(* CODESYS project CoDeSyS_Library_ST_MO
   Author: Razumovskiy
   Company: MechaTronics
   Description: Standart library for main typical devices
   LanguageModelAttribute: qualified-access-only
   Title: mt
   Version: 0.1.0.0

Project tree, tasks and I/O mapping:
  libraries: Standard, * (System)
  Drivers/
    FB_drv/
      function block drv_AI [ST]
      function block drv_AO [ST]
      function block drv_DI [ST]
      function block drv_DO [ST]
      function block drv_DOA [ST]
      function block drv_Flow [ST]
      function block drv_M [ST]
      function block drv_MR [ST]
      function block drv_V [ST]
    FB_sub/
      function sub_Axis_SP [ST]
      function block sub_Calibration [ST]
      function block sub_Filter [ST]
      function block sub_Slow [ST]
    UDT/
      data type AI_cfg
      data type AI_state
      data type AO_cfg
      data type AO_state
      data type Axis_cfg
      data type Axis_state
      data type DI_cfg
      data type DO_cfg
      data type DO_cfg_ext
      data type FE_cfg
      data type FE_state
      data type M_cfg
      data type M_state
      data type sub_Slow_cfg
      data type V_cfg
      data type V_state
    Union/
      uni/
        data type uni_AI_alarm
        data type uni_AI_cfg
        data type uni_AO_cfg
        data type uni_Axis_cfg
        data type uni_Axis_operation
        data type uni_DI_cfg
        data type uni_DO_cfg
        data type uni_FE_cfg
        data type uni_M_alarm
        data type uni_M_cfg
        data type uni_sub_Slow
        data type uni_V_alarm
        data type uni_V_cfg
      uni_udt/
        data type udt_AI_alarm
        data type udt_AI_cfg
        data type udt_AO_cfg
        data type udt_Axis_cfg
        data type udt_Axis_ErrorID
        data type udt_Axis_operation
        data type udt_DI_cfg
        data type udt_DO_cfg
        data type udt_FE_cfg
        data type udt_M_alarm
        data type udt_M_cfg
        data type udt_sub_Slow
        data type udt_V_alarm
        data type udt_V_cfg
  global variables sys
  System/
    FC/
      function drv_Alarm [ST]
      function drv_CMD [ST]
      function drv_Converter [ST]
      function drv_Scale [ST]
      function drv_Time_01S [ST]
      function drv_Time_C [ST]
      function drv_Time_R [ST]
      function drv_Time_S [ST]
      function drv_Time_X [ST]
    List/
      data type list_AI_SP
      data type list_Axis_SP
      data type list_Range
    UDT/
      data type Time_C
      data type Time_R
      data type Time_S
      data type Time_X
      data type udt_CMD
      data type udt_dev_list
      data type udt_DTL
      data type udt_state
      data type udt_Timer
      data type uni_CMD
      data type uni_dev_list
      data type uni_state
      data type uni_Timer
    program x00_Start [ST]
    program x99_End [ST]
  Информация библиотеки/
    function GetLibVersion [ST]
    function GetLibVersionNumber [ST]
    function IsLibReleased [ST]
*)

// Drivers/UDT/AI_cfg
TYPE AI_cfg :
STRUCT
	//configuration struct for Analog Inputs
		cfg				:uni_AI_cfg;	// HMI 0:	configuration word
		Input_Type		:INT := 1;		// HMI 1:	Input type: 0 = 0..20, 1 = 4..20, 2 = 0..10, 3 = Pt100, 4 = Pt1000
		Value_Type		:INT := 0;		// HMI 2:	Value type: 0 = %, 1 = Hz, 2 = l/h, etc
		Filter_Type		:INT := 1;		// HMI 3:	Execution clock for filter: 0 = every cycle of PLC, 1 = 0.1s, 2 = 1s
		Filter_Lim		:INT := 100;	// HMI 4:	Value of records in filter buffer
		Range			:list_Range;	// HMI 5:	Singal scale range
		Calibration		:REAL;			// HMI 13:	Static correction
		Multiplier		:REAL := 1;		// HMI 15:	Multiple correction
		SP				:list_AI_SP;	// HMI 17:	SP for limits
		T_SP			:ARRAY [0..3] OF INT;// HMI 26:	SP timers for limits
		ID				:INT;			// HMI 30:	ID for SCADA
		Name			:ARRAY [0..9] OF BYTE; // HMI 31:	Name
		ADDR			:INT;			// PLC xx:	address of inputs
		// HMI x - x is word number in shift address by start address
END_STRUCT
END_TYPE

// Drivers/UDT/AI_state
TYPE AI_state :
STRUCT
	//condition for Analog Inputs
		state		:uni_state;			// PLC 0:	condition word
		alarm		:uni_AI_alarm;		// HMI 1:	alarm word
		Status		:INT;				// HMI 2:	Status code for HMI
		Result		:REAL;				// HMI 3:	Result of convertation
		Signal		:REAL;				// HMI 5:	Input signal
		(*
			0 - disable
			1 - Result > L and Result < H
			2 - Result < L and Result > LL
			3 - Result > H and Result < HH
			4 - alarm "ST"
			5 - alarm "NC"
			6 - alarm LL
			7 - alarm HH
			
			if any alarm, than HMI will send message
		*)
END_STRUCT
END_TYPE

// Drivers/UDT/AO_cfg
TYPE AO_cfg :
STRUCT
	//configuration struct for Analog Outputs
		cfg				:uni_AO_cfg;	// HMI 0:	configuration word
		Output_Type		:INT := 1;		// HMI 1:	Output type: 0 = 0..20, 1 = 4..20, 2 = 0..10, 3 = Pt100, 4 = Pt1000
		Value_Type		:INT := 0;		// HMI 2:	Value type: 0 = %, 1 = Hz, 2 = l/h, etc
		Range			:list_Range;	// HMI 3:	Singal scale range
		SP_M			:REAL;			// HMI 10:	SP in manual mode
		ID				:INT;			// HMI 11:	ID for SCADA
		Name			:ARRAY [0..9] OF BYTE; // HMI 12:	Name
		ADDR			:INT;			// PLC xx:	address of inputs
END_STRUCT
END_TYPE

// Drivers/UDT/AO_state
TYPE AO_state :
STRUCT
	//condition for Analog Inputs
		state		:uni_state;			// HMI 0:	condition word
		Status		:INT;				// HMI 1:	Status code for HMI
		Result		:REAL;				// HMI 2:	Result of convertation
		Signal		:REAL;				// HMI 4:	Input signal
		(*
			0 - disable
			1 - activate
			
			if any alarm, than HMI will send message
		*)
END_STRUCT
END_TYPE

// Drivers/UDT/Axis_cfg
TYPE Axis_cfg :
STRUCT
	//configuration struct for Analog Inputs
		cfg				:uni_Axis_cfg;	// HMI 0:	configuration word
		Mode			:INT;			//	режим работы
		listSP			:list_Axis_SP;	//  уставки перемещения
		Direction		:BYTE := 1;
		posHome			:LREAL := 0.0;	//	уставка положения при калибровке нулевой точки
		ID				:INT;			// HMI 28:	ID for SCADA
		Name			:ARRAY [0..9] OF BYTE; // HMI 29:	Name
END_STRUCT
END_TYPE

// Drivers/UDT/Axis_state
TYPE Axis_state :
STRUCT
	//condition for Analog Inputs
		state		:uni_state;		// PLC 0:	condition word
		error		:uni_Axis_operation;// HMI 1:	alarm word
		busy		:uni_Axis_operation;
		done		:uni_Axis_operation;
		valid		:uni_Axis_operation;
		abort		:uni_Axis_operation;
		errorID		:udt_Axis_ErrorID;
		Status		:INT;				// HMI 2:	Status code for HMI
		Error_ID	:DWORD;				// HMI 3:	ErrorID
		Position	:LREAL;				// HMI 5:	Actual position
END_STRUCT
END_TYPE

// Drivers/UDT/DI_cfg
TYPE DI_cfg :
STRUCT
	cfg					:uni_DI_cfg;	// HMI 0:	configuration word
	//SP and another settings for Discrete Inputs
		SP_T_ON			:INT;			// HMI 1:	SP Time chatter filter starting, seconds
		SP_T_OFF		:INT;			// HMI 2:	SP Time chatter filter before stoping, seconds
END_STRUCT
END_TYPE

//History log:
//2023.01.10
//	1) data type 'bit' -> 'bool'
//	2) delete memory optimisation

// Drivers/UDT/DO_cfg
TYPE DO_cfg :
STRUCT
	cfg					:uni_DO_cfg;	// HMI 0:	configuration word
END_STRUCT
END_TYPE

// Drivers/UDT/DO_cfg_ext
TYPE DO_cfg_ext :
STRUCT
	cfg					:uni_DO_cfg;	// HMI 0:	configuration word
	//SP and another settings for Discrete Outputs
		SP_T			:REAL;			// HMI 1:	SP Time for impulse or PWM mode
		SP_A			:REAL;			// PLC 3:	SP % for PWM mode in auto mode
		SP_M			:REAL;			// PLC 5:	SP % for PWM mode in Manual mode
		SP_Min			:REAL := 10;	// PLC 7:	SP minimum value for switch on
		SP_Max			:REAL := 90;	// PLC 9:	SP value, while not switch off
END_STRUCT
END_TYPE

// Drivers/UDT/FE_cfg
TYPE FE_cfg :
STRUCT
	//configuration struct for FlowMeter
		cfg				:uni_FE_cfg;	// HMI 0:	configuration word
		Wieght			:REAL := 0.1;	// HMI 1:	Weight for 1 impulse
		Size_Wieght		:INT := 0;		// HMI 3:	Wieght of control unit - ml, l, m3
		Size_Time		:INT;			// HMI 5:	Speed of flow size: 0 - hour, 1 - minute, 2 - second
		Filter_Lim		:INT := 10;		// HMI 6:	Filter limit for summ values, max = 100
		Filter_Type		:INT;			// HMI 7:	Execution clock for filter: 0 = every cycle of PLC, 1 = 0.1s, 2 = 1s
		Clock			:INT := 1;		// HMI 8:	Cycle time for POU mode, ms
		Seans			:REAL;			// HMI 9:	Last seans data
		PreSP			:REAL;			// HMI 11:	PreSetpoint for one seans control
		SP				:REAL := 1;		// HMI 13:	Setpoint for one seans control
		DB				:REAL := 0.1;	// HMI 15:	Deadband for setpoint
		ID				:INT;			// HMI 17:	ID for SCADA
		Name			:ARRAY [0..9] OF BYTE; // HMI 18:	Name
		ADDR			:INT;			// PLC xx:	address of inputs
END_STRUCT
END_TYPE

// Drivers/UDT/FE_state
TYPE FE_state :
STRUCT
	//condition for Analog Inputs
		state		:uni_state;			// HMI 0:	condition word
		Status		:INT;				// HMI 1:	Status code for HMI
		Result		:REAL;				// HMI 2:	Actual flow speed
		AP			:REAL;				// HMI 4:	Actual flow value
		Last_AP		:REAL;				// HMI 6:	Last flow value
		(*
			0 - disable
			1 - Result > L and Result < H
			2 - Result < L and Result > LL
			3 - Result > H and Result < HH
			4 - alarm "ST"
			5 - alarm "NC"
			6 - alarm LL
			7 - alarm HH
			
			if any alarm, than HMI will send message
		*)
END_STRUCT
END_TYPE

// Drivers/UDT/M_cfg
TYPE M_cfg :
STRUCT
	cfg					:uni_M_cfg;		// HMI 0:	configuration word
	//SP and another settings for Motors
		SP_T_Delay_ON	:INT;			// HMI 1:	SP Time delay before starting, seconds
		SP_T_Delay_OFF	:INT;			// HMI 2:	SP Time delay before stoping, seconds
		SP_T_ON			:INT := 2;		// HMI 3:	SP Time feedback control during start, seconds
		SP_T_OFF		:INT := 2;		// HMI 4:	SP Time feedback control during stop, seconds
		ID				:INT;			// HMI 5:	ID for SCADA
		Name			:ARRAY [0..9] OF BYTE; // HMI 6:	Name
END_STRUCT
END_TYPE

//History log:
//2023.01.11
//	1) data type 'bit' -> 'bool'
//2023.01.18
//	1) delete service interval

// Drivers/UDT/M_state
TYPE M_state :
STRUCT
	state				:uni_state;			// HMI 0:	universal state word
	Alarm				:uni_M_alarm;		// HMI 1:	alarm word for Motors
	//specified condition for Motors	
		Status			:INT;				// HMI 2:	Status code for HMI
		(*
			0 - Successfully stopped
			1 - Successfully started
			2 - In the process of stopping
			3 - In the process of starting
			4 - Service maintance
			5 - alarm "No Ready"
			6 - alarm when stopping / now ON
			7 - alarm when starting / now OFF
			8 - alarm TS
			9 - alarm SF
			10 - alarm communication
			11 - External alarm
			99 - Emergency stop
			
			if any alarm, than device will try to stop
		*)
END_STRUCT
END_TYPE

//History log:
//2023.01.11
//	1) data type 'bit' -> 'bool'

// Drivers/UDT/sub_Slow_cfg
TYPE sub_Slow_cfg :
STRUCT
	cfg					:uni_sub_Slow;	// HMI 0:	configuration word
	//SP and another settings for sub driver Slow
		SP_Min			:REAL;
		SP_Max			:REAL;
		SP_Step_Up		:REAL;
		SP_Step_Down	:REAL;
		SP_T_Up			:REAL;
		SP_T_Down		:REAL;
END_STRUCT
END_TYPE

// Drivers/UDT/V_cfg
TYPE V_cfg :
STRUCT
	cfg					:uni_V_cfg;		// HMI 0:	configuration word
	//SP and another settings for Valves
		SP_T_Delay_ON	:INT;			// HMI 1:	SP Time delay before starting, seconds
		SP_T_Delay_OFF	:INT;			// HMI 2:	SP Time delay before stoping, seconds
		SP_T_ON			:INT := 10;		// HMI 3:	SP Time feedback control during start, seconds
		SP_T_OFF		:INT := 10;		// HMI 4:	SP Time feedback control during stop, seconds
		ID				:INT;			// HMI 5:	ID for SCADA
		Name			:ARRAY [0..9] OF BYTE; // HMI 6:	Name

END_STRUCT
END_TYPE

//History log:
//2023.01.13
//	1) data type 'bit' -> 'bool'
//	2) add TS, SF, SRV, Ext configurations
//	3) add SP_T_KM, fixed default SP time SP_T_ON/OFF '2 -> 10'

// Drivers/UDT/V_state
TYPE V_state :
STRUCT
	state				:uni_state;			// HMI 0:	universal state word
	Alarm				:uni_V_alarm;		// HMI 1:	alarm word for Valves
	//specified condition for Valves
		Status		:INT;					// HMI 2:	Status code for HMI
		(*
			0 - Successfully stopped
			1 - Successfully started
			2 - In the process of stopping
			3 - In the process of starting
			4 - Service maintance
			5 - alarm "No Ready"
			6 - alarm when opening / now ON
			7 - alarm when closing / now OFF
			8 - alarm TS
			9 - alarm SF
			10 - alarm communication
			11 - External alarm
			12 - alarm while opening / now close
			13 - alarm while opening / now no FB
			14 - alarm while closing / now open
			15 - alarm while closing / now no FB
			99 - Emergency stop
			
			if any alarm, than device will try to stop
		*)
END_STRUCT
END_TYPE

//History log:
//2023.01.11
//	1) data type 'bit' -> 'bool'

// System/List/list_AI_SP
TYPE list_AI_SP :
STRUCT
	HH			:REAL := 90;
	H			:REAL := 75;
	L			:REAL := 25;
	LL			:REAL := 10;
	SC			:REAL := 105;
	NC			:REAL := -5;
END_STRUCT
END_TYPE

// System/List/list_Axis_SP
TYPE list_Axis_SP :
STRUCT
	//configuration struct for axis movement
		Position				:LREAL := 0;	//Положение
		Velocity				:LREAL := 10;	//Скорость
		Acceleration			:LREAL := 10;	//Ускорение
		Deceleration			:LREAL := 10;	//Замедление
		C						:LREAL := 1;	//Коэффициент преобразования
END_STRUCT
END_TYPE

// System/List/list_Range
TYPE list_Range :
STRUCT
	Min_In		:REAL := 0;
	Max_In		:REAL := 100;
	Min_Out		:REAL := 0;
	Max_Out		:REAL := 100;
END_STRUCT
END_TYPE

// System/UDT/Time_C
TYPE Time_C :
STRUCT
	//control struct for a Timer Millisecond or counting
		CMD			:uni_Timer;		//command word
		SP			:REAL := 2.0;	//set point
		AP			:REAL;			//actual point
		One			:REAL := 0.1;	//impulse weight
		Percent		:REAL;			//progress 0..100%
		PT			:R_TRIG;		//control of a positive signal front
END_STRUCT
END_TYPE

// System/UDT/Time_R
TYPE Time_R :
STRUCT
	//control struct for a Timer High Accucary
		CMD			:uni_Timer;		//command word
		SP			:REAL := 2.000;	//set point as second
		AP			:REAL;			//actual point	
		RTC			:UDINT;			//real time stamp
		Delta		:UDINT;			//delta time control
		Percent		:REAL;			//progress 0..100%
END_STRUCT
END_TYPE

// System/UDT/Time_S
TYPE Time_S :
STRUCT
	//control struct for a Timer Second
		CMD			:uni_Timer;		//command word
		SP			:INT := 2;		//set point
		AP			:INT;			//actual point	
END_STRUCT
END_TYPE

// System/UDT/Time_X
TYPE Time_X :
STRUCT
	//control struct for a Timer High Accucary
		CMD			:uni_Timer;		//command word
		AP			:REAL;			//actual point	
		RTC			:UDINT;			//real time stamp
		Delta		:UDINT;			//delta time control
END_STRUCT
END_TYPE

// System/UDT/udt_CMD
TYPE udt_CMD :
STRUCT
	//standart control word
		Start_A 	:BIT;		// 0:	command for automatic control
		Start_M 	:BIT;		// 1:	command for manual control
		Manual		:BIT;		// 2:	mode of control (0 - automatic, 1 - manual (user or HMI))
		Lock		:BIT;		// 3:	technological lock
		Force		:BIT;		// 4:	forced control in manual mode
		Service		:BIT;		// 5:	activate service mode
		Local		:BIT;		// 6: 	activate local mode (0 - controlled by PLC, 1 - controlled by local keys)
		Reset		:BIT;		// 7:	resetting of device
		Alarm		:BIT;		// 8:	the device is in the alarm
		ResetOT		:BIT;		// 9:	reset opreational time
		Direction	:BIT;		// 10:	direction of moving
		LowSpeed	:BIT;		// 11:	low speed mode
		Test		:BIT;		// 12:	test run for once
		//you add more configuration bits for the project, if necessary, but not more than 15
END_STRUCT
END_TYPE

// System/UDT/udt_dev_list
TYPE udt_dev_list :
STRUCT
	//general types
		xDI		:BIT;		// 0:	any discrete input in *** mode or state
		xDO		:BIT;		// 1:	any discrete optput in *** mode or state
		xAI		:BIT;		// 2:	any analog input in *** mode or state
		xAO		:BIT;		// 3:	any analog ouput in *** mode or state
		xM		:BIT;		// 4:	any device type "M" in *** mode or state
		xV		:BIT;		// 5:	any device type "V" in *** mode or state
		xAxis	:BIT;		// 6:	any axis in *** mode or state
		Logick	:BIT;		// 7:	any logical block in *** mode or state
		xAny	:BIT;		// 8:	something input/output or device in *** mode or state
		xFE		:BIT;		// 9:	any flowmeter in *** mode or state
END_STRUCT
END_TYPE

// System/UDT/udt_DTL
TYPE udt_DTL :
STRUCT
	//Data Time List
		Year			:UINT;
		Month			:UINT;
		Day				:UINT;
		Hour			:UINT;
		Minute			:UINT;
		Second			:UINT;
		Millisecond		:UINT;
		WeekDay			:UINT;
		WeekYear		:UINT;
END_STRUCT
END_TYPE

// System/UDT/udt_state
TYPE udt_state :
STRUCT
	//unviversal condition word for any devices
		xON				:BIT;		// 0:	device succesfully started and working now
		xOFF			:BIT;		// 1:	device succesfulle stoped and stoping now
		Alarm			:BIT;		// 2:	device in something alarm
		Local			:BIT;		// 3:	device in local mode
		Service			:BIT;		// 4:	device in service mode
		warn_OT			:BIT;		// 5:	warning "Service maintenance is required, the interservice interval is exceeded"
		Pos_Ok			:BIT;		// 6:	position/speed reached or run now
		Ready			:BIT;		// 7:	device ready to start		
		Busy			:BIT;		// 8:	device busy and working now
		Done			:BIT;		// 9:	device finished task
		Enable			:BIT;		//10:	device enabled
		//you may add more configuration bits for the project, if necessary, but not more than 15
END_STRUCT
END_TYPE

// System/UDT/udt_Timer
TYPE udt_Timer :
STRUCT
	//configuration word for Timers
		Start		:BIT;			// 0:	Starting command
		Q			:BIT;			// 1:	Quit
		Pause		:BIT;			// 2:	Pause
		Reset		:BIT;			// 3:	Reset actual point to zero
		SFC			:BIT;			// 4:	Signal front control
		//you add more configuration bits for the project, if necessary, but not more than 16
END_STRUCT
END_TYPE

// System/UDT/uni_CMD
TYPE uni_CMD :
UNION
	//configuration word for Command Word
		hmi		:WORD;			//word for communication
		plc		:udt_CMD;	//tags for programming
END_UNION
END_TYPE

// System/UDT/uni_dev_list
TYPE uni_dev_list :
UNION
	//alarm word for device list
		hmi		:WORD;			//word for communication
		plc		:udt_dev_list;	//tags for programming
END_UNION
END_TYPE

// System/UDT/uni_state
TYPE uni_state :
UNION
	//universal state word
		hmi		:WORD;			//word for communication
		plc		:udt_state;		//tags for programming
END_UNION
END_TYPE

// System/UDT/uni_Timer
TYPE uni_Timer :
UNION
	//alarm word for Timers
		hmi		:WORD;			//word for communication
		plc		:udt_Timer;		//tags for programming
END_UNION
END_TYPE

// Drivers/Union/uni/uni_AI_alarm
TYPE uni_AI_alarm :
UNION
	//alarm word for Analog Inputs
		hmi		:WORD;			//word for communication
		plc		:udt_AI_alarm;	//tags for programming
END_UNION
END_TYPE

// Drivers/Union/uni/uni_AI_cfg
TYPE uni_AI_cfg :
UNION
	//configuration word for Analog Inputs
		hmi		:WORD;			//word for communication
		plc		:udt_AI_cfg;	//tags for programming
END_UNION
END_TYPE

// Drivers/Union/uni/uni_AO_cfg
TYPE uni_AO_cfg :
UNION
	//configuration word for Analog Inputs
		hmi		:WORD;			//word for communication
		plc		:udt_AO_cfg;	//tags for programming
END_UNION
END_TYPE

// Drivers/Union/uni/uni_Axis_cfg
TYPE uni_Axis_cfg :
UNION
	//configuration word forAxis
		hmi		:WORD;			//word for communication
		plc		:udt_Axis_cfg;	//tags for programming
END_UNION
END_TYPE

// Drivers/Union/uni/uni_Axis_operation
TYPE uni_Axis_operation :
UNION
	//modes word for Axis
		hmi		:WORD;			//word for communication
		plc		:udt_Axis_operation;	//tags for programming
END_UNION
END_TYPE

// Drivers/Union/uni/uni_DI_cfg
TYPE uni_DI_cfg :
UNION
	//configuration word for Discrete Inputs
		hmi		:WORD;			//word for communication
		plc		:udt_DI_cfg;	//tags for programming
END_UNION
END_TYPE

// Drivers/Union/uni/uni_DO_cfg
TYPE uni_DO_cfg :
UNION
	//configuration word for Discrete Outputs
		hmi		:WORD;			//word for communication
		plc		:udt_DO_cfg;	//tags for programming
END_UNION
END_TYPE

// Drivers/Union/uni/uni_FE_cfg
TYPE uni_FE_cfg :
UNION
	//configuration word for Analog Inputs
		hmi		:WORD;			//word for communication
		plc		:udt_FE_cfg;	//tags for programming
END_UNION
END_TYPE

// Drivers/Union/uni/uni_M_alarm
TYPE uni_M_alarm :
UNION
	//alarm word for Motors
		hmi		:WORD;			//word for communication
		plc		:udt_M_alarm;	//tags for programming
END_UNION
END_TYPE

// Drivers/Union/uni/uni_M_cfg
TYPE uni_M_cfg :
UNION
	//configuration word for Motors
		hmi		:WORD;			//word for communication
		plc		:udt_M_cfg;		//tags for programming
END_UNION
END_TYPE

// Drivers/Union/uni/uni_sub_Slow
TYPE uni_sub_Slow :
UNION
	//configuration word for sub driver Slow
		hmi		:WORD;			//word for communication
		plc		:udt_sub_Slow;	//tags for programming
END_UNION
END_TYPE

// Drivers/Union/uni/uni_V_alarm
TYPE uni_V_alarm :
UNION
	//alarm word for Valves
		hmi		:WORD;			//word for communication
		plc		:udt_V_alarm;	//tags for programming
END_UNION
END_TYPE

// Drivers/Union/uni/uni_V_cfg
TYPE uni_V_cfg :
UNION
	//configuration word for Valves
		hmi		:WORD;			//word for communication
		plc		:udt_V_cfg;		//tags for programming
END_UNION
END_TYPE

// Drivers/Union/uni_udt/udt_AI_alarm
TYPE udt_AI_alarm :
STRUCT
	//alarm word for Analog Inputs
		alm_ST		:BIT;		// 0:	alarm "No Ready" 
		alm_HH		:BIT;		// 1:	alarm "High alarm level"
		alm_H		:BIT;		// 2:	warning "High work level"
		alm_L		:BIT;		// 3:	warning "Low work level"
		alm_LL		:BIT;		// 4:	alarm "Low alarm level"
		alm_NC		:BIT;		// 5:	alarm "No connect"
		alm_SC		:BIT;		// 6:	alarm "Overload"
		//you add more configuration bits for the project, if necessary, but not more than 16
END_STRUCT
END_TYPE

// Drivers/Union/uni_udt/udt_AI_cfg
TYPE udt_AI_cfg :
STRUCT
	//configuration word for Analog Inputs
		use_Sim		:BIT;			// PLC 0:	0 - Normal mode of operation, 	1 - Simulation mode
		use_NoEmrg	:BIT;			// PLC 1:	0 - Use Emergency signal,		1 - Ignore Emergency signal
		use_RTD		:BIT := FALSE;	// HMI 2:	Use mode RTD/TC scaling
		use_Filter	:BIT := TRUE;	// HMI 3:	Use filter
		use_Light	:BIT;			// HMI 4:	Lighting status for screen indication
		use_Low		:BIT := TRUE;	// PLC 5:	Enable low level alarms
		use_High	:BIT := TRUE;	// PLC 6:	Enable high level alarms
		use_SC		:BIT;			// HMI 7:	use control wire break
		//you add more configuration bits for the project, if necessary, but not more than 16
END_STRUCT
END_TYPE

// Drivers/Union/uni_udt/udt_AO_cfg
TYPE udt_AO_cfg :
STRUCT
	//configuration word for Analog Outputs
		use_Sim		:BIT;			// PLC 0:	0 - Normal mode of operation, 	1 - Simulation mode
		use_NoEmrg	:BIT;			// HMI 1:	0 - Use Emergency signal,		1 - Ignore Emergency signal
		use_Light	:BIT;			// HMI 3:	Lighting status for screen indication
		//you add more configuration bits for the project, if necessary, but not more than 16
END_STRUCT
END_TYPE

// Drivers/Union/uni_udt/udt_Axis_cfg
TYPE udt_Axis_cfg :
STRUCT
	//configuration word for Analog Inputs
		use_Sim		:BIT;			// PLC 0:	0 - Normal mode of operation, 	1 - Simulation mode
		use_NoEmrg	:BIT;			// PLC 1:	0 - Use Emergency signal,		1 - Ignore Emergency signal
		use_Axis	:BIT;			// PLC 2: 	0 - Disable axis,				1 - Enable axis
		set_zero	:BIT;			// PLC 3:	0 - no activities,				1 - Set actual position as ZERO
		//you add more configuration bits for the project, if necessary, but not more than 16
END_STRUCT
END_TYPE

// Drivers/Union/uni_udt/udt_Axis_ErrorID
TYPE udt_Axis_ErrorID :
STRUCT
	//busy word for Axis
		read_position		:DWORD;		// 0:	MC_Position
		read_error			:DWORD;		// 1:	MC_ReadError
		reset_axis			:DWORD;		// 2:	MC_Reset
		power_on			:DWORD;		// 3:	MC_Power
		move_home			:DWORD;		// 4:	MC_Home
		move_jog			:DWORD;		// 5:	MC_Jog
		move_abs			:DWORD;		// 5:	MC_Abs
		move_vel			:DWORD;		// 7:	MC_Velocity
		set_pos				:DWORD;		// 8:	MC_SetPos
		tmp					:DWORD;		// 9:	temp value
		//you may add more configuration bits for the project, if necessary, but not more than 15
END_STRUCT
END_TYPE

// Drivers/Union/uni_udt/udt_Axis_operation
TYPE udt_Axis_operation :
STRUCT
	//busy word for Axis
		read_position		:BIT;		// 0:	MC_Position
		read_error			:BIT;		// 1:	MC_ReadError
		reset_axis			:BIT;		// 2:	MC_Reset
		power_on			:BIT;		// 3:	MC_Power
		move_home			:BIT;		// 4:	MC_Home
		move_jog			:BIT;		// 5:	MC_Jog
		move_abs			:BIT;		// 6:	MC_Abs
		move_vel			:BIT;		// 7:	MC_Velocity
		set_pos				:BIT;		// 8:	MC_SetPos
		ext					:BIT;		// 9:	external value
		tmp					:BIT;		//10:	temp value
		//you may add more configuration bits for the project, if necessary, but not more than 15
END_STRUCT
END_TYPE

// Drivers/Union/uni_udt/udt_DI_cfg
TYPE udt_DI_cfg :
STRUCT
	//configuration struct for Discrete Inputs
		use_Sim			:BIT;			// PLC 0:	0 - Normal mode of operation, 	1 - Simulation mode
		use_NoEmrg		:BIT;			// HMI 1:	0 - Use Emergency signal,		1 - Ignore Emergency signal
		use_NC			:BIT;			// HMI 2:	0 - Normal Open Signal, 		1 - Normal Close Signal
		use_Filter		:BIT;			// HMI 3:	0 - Not use filter,				1 - Use chatter filter
		//you may add more configuration bits for the project, if necessary, but not more than 15
END_STRUCT
END_TYPE

// Drivers/Union/uni_udt/udt_DO_cfg
TYPE udt_DO_cfg :
STRUCT
	//configuration struct for Discrete Outputs
		use_Sim			:BIT;			// PLC 0:	0 - Normal mode of operation, 	1 - Simulation mode
		use_NoEmrg		:BIT;			// HMI 1:	0 - Use Emergency signal,			1 - Ignore Emergency signal
		use_NC			:BIT;			// HMI 2:	0 - Normal Open Signal, 			1 - Normal Close Signal
		use_Impulse		:BIT;			// HMI 3:	0 - Permanent mode of operation, 	1 - Impulse mode of operation
		use_PWM			:BIT;			// HMI 4:	0 - Constant signal,				1 - PWM signal
		//you may add more configuration bits for the project, if necessary, but not more than 15
END_STRUCT
END_TYPE

// Drivers/Union/uni_udt/udt_FE_cfg
TYPE udt_FE_cfg :
STRUCT
	//configuration word for Analog Inputs
		use_Sim		:BIT;			// PLC 0:	0 - Normal mode of operation, 	1 - Simulation mode
		use_NoEmrg	:BIT;			// PLC 1:	0 - Use Emergency signal,		1 - Ignore Emergency signal
		use_POU		:BIT;			// HMI 2:	Call FE in special POU with fixed time
		use_Filter	:BIT := TRUE;	// HMI 3:	Use filter
		use_Light	:BIT;			// HMI 4:	Lighting status for screen indication
		use_DI		:BIT;			// HMI 5:	Use DI signal
		use_FM		:BIT;			// HMI 6:	Use weight control
		use_FM_Add	:BIT;			// HMI 7:	Use add weight control
		use_PreSP	:BIT := TRUE;	// HMI 8:	Use pre-SP  control
		use_SP		:BIT := TRUE;	// HMI 9:	Use SP control
		//you add more configuration bits for the project, if necessary, but not more than 16
END_STRUCT
END_TYPE

// Drivers/Union/uni_udt/udt_M_alarm
TYPE udt_M_alarm :
STRUCT
	//alarm word for Motors
		alm_QF			:BIT;		// 0:	alarm "No Ready" 
		alm_Start		:BIT;		// 1:	alarm "No In Work when starting"
		alm_Stop		:BIT;		// 2:	alarm "In Work when stopping"
		alm_TS			:BIT;		// 3:	alarm "No TS"
		alm_SF			:BIT;		// 4:	alarm "No Safety Signal"
		alm_Ext			:BIT;		// 5:	alarm "External alarm"
		alm_Link		:BIT;		// 6:	alarm communication
		alm_ES			:BIT;		// 7:	alarm "Emergency Stop"
		//you may add more configuration bits for the project, if necessary, but not more than 15
END_STRUCT
END_TYPE

// Drivers/Union/uni_udt/udt_M_cfg
TYPE udt_M_cfg :
STRUCT
	//configuration word for Motors
		use_Sim			:BIT;			// HMI 0:	0 - Normal mode of operation,	1 - Simulation mode
		use_NoEmrg		:BIT;			// HMI 1:	0 - Use Emergency signal,		1 - Ignore Emergency signal
		use_QF			:BIT := TRUE;	// HMI 2:	Feedback control "Ready"
		use_KM			:BIT := TRUE;	// HMI 3:	Feedback control "In work"
		use_Signal 		:BIT := TRUE;	// HMI 4:	Use external REQ
		//you may add more configuration bits for the project, if necessary, but not more than 15
END_STRUCT
END_TYPE

// Drivers/Union/uni_udt/udt_sub_Slow
TYPE udt_sub_Slow :
STRUCT
	//configuration struct for sub driver Slow
		//configuration word for Valves
		Enable			:BIT;			// HMI 0:	Enable algorythm
		use_Up			:BIT;			// HMI 1:	use slow mode for up value
		use_Down		:BIT;			// HMI 2:	use slow mode for down value
		use_Force_Up	:BIT;			// HMI 3:	use force mode for first up
		use_Force_Down	:BIT;			// HMI 4:	use force mode for last down
END_STRUCT
END_TYPE

// Drivers/Union/uni_udt/udt_V_alarm
TYPE udt_V_alarm :
STRUCT
	//alarm word for Valves
		alm_QF			:BIT;		// 0:	alarm "No Ready" 
		alm_Open		:BIT;		// 1:	alarm while opening
		alm_Close		:BIT;		// 2:	alarm while closing
		alm_Duo			:BIT;		// 3:	alarm duo signals FB_Open and FB_Close at once
		alm_TS			:BIT;		// 4:	alarm "No TS"
		alm_Ext			:BIT;		// 5:	alarm "External alarm"
		alm_Link		:BIT;		// 6:	alarm communication
		alm_ES			:BIT;		// 7:	alarm "Emergency Stop"
		//you may add more configuration bits for the project, if necessary, but not more than 15
END_STRUCT
END_TYPE

// Drivers/Union/uni_udt/udt_V_cfg
TYPE udt_V_cfg :
STRUCT
	//configuration struct for Valves
		//configuration word for Valves
		use_Sim			:BIT;			// HMI 0:	0 - Normal mode of operation,	1 - Simulation mode
		use_NoEmrg		:BIT;			// HMI 1:	0 - Use Emergency signal,		1 - Ignore Emergency signal
		use_QF			:BIT := TRUE;	// HMI 2:	Feedback control "Ready"
		use_FB_Open		:BIT := TRUE;	// HMI 3:	Feedback control "Valve Opened"
		use_FB_Close	:BIT := TRUE;	// HMI 4:	Feedback control "Valve Closed"
		use_CWF			:BIT := TRUE;	// HMI 5:	Close While Fault
		use_Air			:BIT;			// HMI 6:	Work mode for air valves
		use_Duo			:BIT;			// HMI 7:	Work mode for CW/CCW
		use_Once		:BIT;			// HMI 8:	Work mode without open/close feedback control after finishing movement
		use_Signal 		:BIT := TRUE;	// HMI 9:	Use external REQ
END_STRUCT
END_TYPE

// sys
{attribute 'qualified_only'}
VAR_GLOBAL
	//General management
		//Global controls
			All_Block		AT %MX0.0	:BOOL;				//Emergency stop
			All_Reset		AT %MX0.1	:BOOL;				//Reset all alarms
			All_Sim			AT %MX0.2	:BOOL;				//Switch simulation mode for all devices
			All_Auto		AT %MX0.3	:BOOL;				//Reset "CMD.plc.Manual" for all devices
			Silence			AT %MX0.4	:BOOL;				//Disable siren from HMI
			Save			AT %MX0.5	:BOOL;				//Save data to PVL
		//Service tags
			alm				AT %MW1		:uni_dev_list;		//Alarms flags for devices
			man				AT %MW2		:uni_dev_list;		//Manual flags for devices
			sim				AT %MW3		:uni_dev_list;		//Simulation flags for devices
			DTL				:udt_DTL;						//System time
			UpTime			:TIME;							//Work time after power on
			UpTime_ms		:UDINT;							//Work time after power on as millisecond
		//Global data
			LibVersion		AT %ML1		:VERSION;			//Version code
		
		//Additional tags and constans
			second			:REAL := (1.0/3600.0);	//wight of 1 second in hour format
			dev				:INT;					//device counter for FOR
			aws_ON			:BOOL := TRUE;			//always TRUE
			aws_OFF			:BOOL := FALSE;			//always FALSE
			StartUp_Load	:BOOL;		//First load configuration after power on
				
		//Impulse tags
			pulse_01s	:BOOL;					//global trigger 100 ms
			pulse_1s	:BOOL;					//global trigger 1 second
			
		//Clock tags
			clock_01s	:BOOL;					//global clock for 100 ms
			clock_05s	:BOOL;					//global clock for 500 ms
			clock_1s	:BOOL;					//global clock for 1 s
END_VAR

// System/x00_Start
PROGRAM x00_Start
VAR
	pulse_100ms			:UDINT;
	pulse_s				:UDINT;
	clock_100ms			:UDINT;
	clock_500ms			:UDINT;
	clock_s				:UDINT;
	support				:WORD;
	PT					:ARRAY [0..1] OF R_TRIG;
	NT					:ARRAY [0..1] OF F_TRIG;
END_VAR

//Read system time
	sys.UpTime := TIME();
	sys.UpTime_ms := TIME_TO_UDINT(sys.UpTime);
	
//Read library version
	sys.LibVersion := GetLibVersion();

//Pulse generation
	//pulse 100 ms
		IF (sys.UpTime_ms - pulse_100ms) >= 100 THEN
			sys.pulse_01s := TRUE;
			pulse_100ms := sys.UpTime_ms;
		else
			sys.pulse_01s := FALSE;
		END_IF;
	//pulse 1 s
		IF (sys.UpTime_ms - pulse_s) >= 1000 THEN
			sys.pulse_1s := TRUE;
			pulse_s := sys.UpTime_ms;
		else
			sys.pulse_1s := FALSE;
		END_IF;
		
//Clock generation
	//clock 100 ms
		IF (sys.UpTime_ms - clock_100ms) >= 100 THEN
			IF NOT sys.clock_01s THEN
				sys.clock_01s := TRUE;
			ELSE
				sys.clock_01s := FALSE;
			END_IF;
			clock_100ms := sys.UpTime_ms;
		END_IF;
		
	//clock 500 ms
		IF (sys.UpTime_ms - clock_500ms) >= 500 THEN
			IF NOT sys.clock_05s THEN
				sys.clock_05s := TRUE;
			ELSE
				sys.clock_05s := FALSE;
			END_IF;
			clock_500ms := sys.UpTime_ms;
		END_IF;
		
	//clock 1 s
		IF (sys.UpTime_ms - clock_s) >= 1000 THEN
			IF NOT sys.clock_1s THEN
				sys.clock_1s := TRUE;
			ELSE
				sys.clock_1s := FALSE;
			END_IF;
			clock_s := sys.UpTime_ms;
		END_IF;

END_PROGRAM

// Информация библиотеки/GetLibVersion
// This function has been automatically generated from the project information.
FUNCTION GetLibVersion : VERSION
VAR_INPUT
	
END_VAR

GetLibVersion.uiMajor := 0;
GetLibVersion.uiMinor := 1;
GetLibVersion.uiServicePack := 0;
GetLibVersion.uiPatch := 0;

END_FUNCTION

// System/x99_End
PROGRAM x99_End
VAR
END_VAR

//manual signal processing
	IF sys.man.plc.xAI OR sys.man.plc.xAO OR sys.man.plc.xDI OR sys.man.plc.xDO OR sys.man.plc.xM OR sys.man.plc.xV OR sys.man.plc.xAxis THEN
		sys.man.plc.xAny := TRUE;
	ELSE
		sys.man.plc.xAny := FALSE;
	END_IF;

//error signal processing
	IF sys.alm.plc.xAI OR sys.alm.plc.xM  OR sys.alm.plc.xV OR sys.alm.plc.xAxis OR sys.alm.plc.Logick THEN
		sys.alm.plc.xAny := TRUE;
	ELSE
		sys.alm.plc.xAny := FALSE;
	END_IF;
	
//simulation signal processing
	IF sys.sim.plc.xDO OR sys.sim.plc.xAO  OR sys.sim.plc.xM OR sys.sim.plc.xV OR sys.sim.plc.xAxis THEN
		sys.sim.plc.xAny := TRUE;
	ELSE
		sys.sim.plc.xAny := FALSE;
	END_IF;
	
//reset alarm processing
	IF sys.All_Reset THEN
		sys.alm.plc.xDO := FALSE;
		sys.alm.plc.xAO := FALSE;
		sys.alm.plc.xM := FALSE;
		sys.alm.plc.xV := FALSE;
		sys.alm.plc.xAxis := FALSE;
		sys.alm.plc.xAI := FALSE;
		sys.alm.plc.xM := FALSE;
		sys.alm.plc.xV := FALSE;
		sys.alm.plc.Logick := FALSE;
		sys.All_Reset := FALSE;
		sys.Silence := FALSE;
	END_IF;

//reset auto
	IF sys.All_Auto THEN
		sys.man.plc.xAI := FALSE;
		sys.man.plc.xDI := FALSE;
		sys.man.plc.xM := FALSE;
		sys.man.plc.xV := FALSE;
		sys.man.plc.xAO := FALSE;
		sys.man.plc.xDO := FALSE;
		sys.All_Auto := FALSE;
	END_IF
	
//Save data to PVL
	IF sys.Save THEN
		sys.Save := FALSE;
	END_IF

END_PROGRAM

// Информация библиотеки/GetLibVersionNumber
// This function has been automatically generated from the project information.
FUNCTION GetLibVersionNumber : DWORD
VAR_INPUT
	
END_VAR

GetLibVersionNumber := 65536;

END_FUNCTION

// Информация библиотеки/IsLibReleased
// This function has been automatically generated from the project information.
FUNCTION IsLibReleased : BOOL
VAR_INPUT
	
END_VAR

IsLibReleased := FALSE;

END_FUNCTION

// Drivers/FB_drv/drv_AI
FUNCTION_BLOCK drv_AI
VAR_INPUT
	Signal			:REAL;			//Analog input signal from PLC
END_VAR	
VAR_IN_OUT
	CMD				:uni_CMD;		//Non-retain structure with command word
	cfg				:AI_cfg;		//Retain structure with settings
	state			:AI_state;		//Non-retain structure with states information
END_VAR
VAR_OUTPUT
	Result			:REAL;			//Signal from sensor
END_VAR
VAR
	Value			:REAL;			//tmp value for calculating 
	support			:WORD;			//internal command buffer
	alm				:ARRAY [0..3] OF BOOL;			//support word for transfer alarms
	cnt				:INT;			//internal counter
	PT				:ARRAY [0..1] OF R_TRIG;
	NT				:ARRAY [0..1] OF F_TRIG;
	Clock			:ARRAY [0..3] OF Time_S;
	Filter			:sub_Filter;
END_VAR

//ANALOG INPUT
//control of typical analog sensors
// - pressure
// - level
// - flowmeter
// - etc

//global commands
	//auto mode
		IF sys.All_Auto THEN
			CMD.plc.Manual := FALSE;
		END_IF;
	//global reset
		IF sys.All_Reset THEN
			CMD.plc.Reset := TRUE;
		END_IF
		
//convert data
	//input scaling
	drv_Scale(
		Value := Signal,
		Input_Type := cfg.Input_Type,
		Range := cfg.Range,
		Result => state.Signal);
		
//NC control
	IF cfg.Input_Type = 1 AND state.Signal < 2.5 AND cfg.cfg.plc.use_SC AND CMD.plc.Start_A THEN
		state.alarm.plc.alm_NC := TRUE;
	END_IF
	
//SC control
IF cfg.cfg.plc.use_SC AND CMD.plc.Start_A  THEN
	CASE cfg.Input_Type OF 
		0: 	IF state.Signal > 21.0 AND cfg.cfg.plc.use_SC THEN			//0..20 mA
				state.alarm.plc.alm_SC := TRUE;
			END_IF
		1: 	IF state.Signal > 21.0 AND cfg.cfg.plc.use_SC THEN			//4..20 mA
				state.alarm.plc.alm_SC := TRUE;
			END_IF
		2: 	IF state.Signal > 10.5 AND cfg.cfg.plc.use_SC THEN			//0..10 V
				state.alarm.plc.alm_SC := TRUE;
			END_IF
		3: 	IF state.Signal > 155.0 AND cfg.cfg.plc.use_SC THEN			//-150..+150 C
				state.alarm.plc.alm_SC := TRUE;
			END_IF
		4: 	IF state.Signal > 255.0 AND cfg.cfg.plc.use_SC THEN			//-150..+250 C
				state.alarm.plc.alm_SC := TRUE;
			END_IF
	END_CASE
end_if
	
//device control
// 	drv_CMD(Emergency := support.0,
// 			CMD := CMD);
	//manual mode flag
		IF CMD.plc.Manual THEN sys.man.plc.xAI := TRUE; END_IF;
		
//data convert to phisycal value scale
	drv_Converter(
		Signal := Signal,
		Range := cfg.Range,
		Result => Value);
		
//signal's filter
	Filter(
		Start := CMD.plc.Start_A AND cfg.cfg.plc.use_Filter,
		Signal := Value,
		Filter_Type := cfg.Filter_Type,
		Filter_Lim := cfg.Filter_Lim,
		Result => Result);
		
//no filtering mode
	IF NOT cfg.cfg.plc.use_Filter THEN
		Result := Value;
	END_IF
	
//signal's correction
	IF NOT CMD.plc.Start_A THEN
		Result := 0;
	ELSE
		Result := Result * cfg.Multiplier + cfg.Calibration;
	END_IF
	
//state signal transfer
	state.Result := Result;

//alarms without time control
	//ST
		IF state.alarm.plc.alm_NC OR state.alarm.plc.alm_SC AND cfg.cfg.plc.use_SC AND CMD.plc.Start_A THEN
			state.alarm.plc.alm_ST := TRUE;
		END_IF
	
//alarms with time control
	//HH
		drv_Alarm(
			Signal := (Result > cfg.SP.HH AND cfg.cfg.plc.use_High),
			Reset := (CMD.plc.Reset OR NOT CMD.plc.Start_A),
			Clock := Clock[0].CMD,
			Alarm := alm[0]);
		state.alarm.plc.alm_HH := alm[0];
	//H
		drv_Alarm(
			Signal := (Result > cfg.SP.H),
			Reset := (CMD.plc.Reset OR NOT CMD.plc.Start_A OR (Result < cfg.SP.H)),
			Clock := Clock[1].CMD,
			Alarm := alm[1]);
		state.alarm.plc.alm_H := alm[1];
	//L
		drv_Alarm(
			Signal := (Result < cfg.SP.L),
			Reset := (CMD.plc.Reset OR NOT CMD.plc.Start_A OR (Result > cfg.SP.L)),
			Clock := Clock[2].CMD,
			Alarm := alm[2]);
		state.alarm.plc.alm_L := alm[2];
	//LL
		drv_Alarm(
			Signal := (Result < cfg.SP.LL AND cfg.cfg.plc.use_Low),
			Reset := (CMD.plc.Reset OR NOT CMD.plc.Start_A),
			Clock := Clock[3].CMD,
			Alarm := alm[3]);
		state.alarm.plc.alm_LL := alm[3];

//global alarm
	IF (state.alarm.plc.alm_ST OR state.alarm.plc.alm_HH OR state.alarm.plc.alm_LL) AND CMD.plc.Start_A THEN
		state.state.plc.Alarm := TRUE;
		sys.alm.plc.xAI := TRUE;
		CMD.plc.Alarm := TRUE;
	END_IF
	
//reset
	IF CMD.plc.Reset THEN
		state.alarm.hmi := 0;
		FOR cnt := 0 TO 3 DO
			Clock[cnt].CMD.plc.Reset := TRUE;
		END_FOR
		state.alarm.plc.alm_HH := FALSE;
		state.alarm.plc.alm_LL := FALSE;
		state.alarm.plc.alm_SC := FALSE;
		state.alarm.plc.alm_ST := FALSE;
		state.state.plc.Alarm := FALSE;
		CMD.plc.Alarm := FALSE;
		CMD.plc.Reset := FALSE;
	END_IF
	
//global state
	IF CMD.plc.Start_A THEN
		state.state.plc.xON := TRUE;
		state.state.plc.xOFF := FALSE;
	ELSE
		state.state.plc.xON := FALSE;
		state.state.plc.xOFF := TRUE;
	END_IF
	
//HMI light
	IF cfg.cfg.plc.use_Light THEN
		IF CMD.plc.Start_A THEN state.Status := 1; END_IF
		IF NOT state.alarm.plc.alm_L AND NOT state.alarm.plc.alm_H THEN state.Status := 1; END_IF
		IF state.alarm.plc.alm_L AND NOT state.alarm.plc.alm_LL THEN state.Status := 2; END_IF
		IF state.alarm.plc.alm_H AND NOT state.alarm.plc.alm_HH THEN state.Status := 3; END_IF
		IF state.alarm.plc.alm_LL THEN state.Status := 4; END_IF
		IF state.alarm.plc.alm_HH THEN state.Status := 5; END_IF
		IF state.alarm.plc.alm_ST THEN state.Status := 6; END_IF
		IF NOT CMD.plc.Start_A THEN state.Status := 0; END_IF
	ELSE
		state.Status := 0;
	END_IF
	
//call timers
	FOR cnt := 0 TO 3 DO
		Clock[0].SP := cfg.T_SP[cnt];
		drv_Time_S (Clock[cnt]);
	END_FOR

END_FUNCTION_BLOCK

// System/FC/drv_Scale
FUNCTION drv_Scale : bool
VAR_INPUT
	Value			:REAL;			//Analog input signal from PLC
	Input_Type		:INT;			//Input type: 0 = 0..20, 1 = 4..20, 2 = 0..10, 3 = Pt100, 4 = Pt1000
	Range			:list_Range;	//Signal scale range
END_VAR
VAR_OUTPUT
	Result 			:REAL;			//Analog input in phisical value
END_VAR
VAR
	Type_Min		:REAL;			//Minimum limit
	Type_Max		:REAL;			//Maximum limit
	Type_Limit		:int := 4;		//Update type in cyclic
END_VAR

//configuration transfering	
CASE Input_Type OF
	0: Type_Min := 0.0; Type_Max := 20.0;
	1: Type_Min := 4.0; Type_Max := 20.0;
	2: Type_Min := 0.0; Type_Max := 10.0;
	3: Result := Value;
	4: Result := Value;
END_CASE

//calculate real input value
IF Input_Type < 3 THEN
	Result := (Type_Max - Type_Min) / (Type_Limit - 0.0) * Value + Type_Min;
END_IF

//update type in cycle increment
IF Input_Type > Type_Limit THEN Input_Type := 0; END_IF

END_FUNCTION

// System/FC/drv_CMD
FUNCTION drv_CMD : bool
VAR_INPUT
	Emergency		:BOOL;		//signal of All_Block and Safety conditions
END_VAR
VAR_IN_OUT
	CMD				:uni_CMD;	//standart command word
END_VAR

// Device mode determination
	IF NOT Emergency THEN
		//Normal mode
		IF NOT CMD.plc.Force THEN
			//No technological lock
			IF NOT CMD.plc.Lock AND NOT CMD.plc.Alarm AND NOT CMD.plc.Service THEN
				//No manual mode
				IF NOT CMD.plc.Manual THEN
					CMD.plc.Start_M := CMD.plc.Start_A;
				END_IF;
			ELSE
				//Technological lock or device alarm
				CMD.plc.Start_M := FALSE;
			END_IF;
		END_IF;
	ELSE
		//Emergency stop
		CMD.plc.Start_M := FALSE;
	END_IF;

END_FUNCTION

// System/FC/drv_Converter
FUNCTION drv_Converter : bool
VAR_INPUT
	Signal			:REAL;			//Analog input signal from PLC
	Range			:list_Range;	//Signal scale range
END_VAR
VAR_OUTPUT
	Result			:REAL;			//Convertation result
END_VAR
VAR
	inv				:BOOL;			//inverse range
	Range_In		:REAL;			//full input range
	Range_Out		:REAL;			//full value range
	RR_Scale		:REAL;			//range in to range out scale
	Value_Min		:REAL;			//actual minimum output value
	Value_Max		:REAL;			//actual maximum output value
	Buffer			:REAL;			//tmp value for calculating
END_VAR

//Диапазон входного сигнала
IF Range.Min_In >= 0 THEN
    Range_In := Range.Max_In - Range.Min_In;
ELSE
    Range_In := Range.Max_In + ABS(Range.Min_In);
END_IF;

//Диапазон выходного сигнала
inv := FALSE;
IF Range.Min_Out >= 0 AND Range.Max_Out >= 0 THEN
    IF Range.Max_Out > Range.Min_Out THEN
        Range_Out := Range.Max_Out - Range.Min_Out;
        Value_Min := Range.Min_Out;
        Value_Max := Range.Max_Out;
    END_IF;
    IF Range.Max_Out < Range.Min_Out THEN
        Range_Out := Range.Min_Out - Range.Max_Out;
        Value_Min := Range.Max_Out;
        Value_Max := Range.Min_Out;
		inv := TRUE;
    END_IF;
END_IF;
IF Range.Min_Out <= 0 AND Range.Max_Out >= 0 THEN
    Range_Out := Range.Max_Out + ABS(Range.Min_Out);
	Value_Min := Range.Min_Out;
    Value_Max := Range.Max_Out;
END_IF;
IF Range.Min_Out <= 0 AND Range.Max_Out <= 0 THEN
    Range_Out := ABS(Range.Max_Out) + ABS(Range.Min_Out);
	Value_Min := Range.Min_Out;
    Value_Max := Range.Max_Out;
END_IF;
IF Range.Min_Out >= 0 AND Range.Max_Out <= 0 THEN
    Range_Out := ABS(Range.Max_Out) + ABS(Range.Min_Out);
	Value_Min := Range.Max_Out;
    Value_Max := Range.Min_Out;
END_IF;

//Соотношение диапазонов
IF Range_Out <> 0 THEN
	RR_Scale := Range_In / Range_Out;
END_IF

//Линеаризация
IF RR_Scale <> 0 THEN
	Buffer := Signal / RR_Scale;
END_IF

//Коррекция
Buffer := Buffer + Value_Min;

//Инверсия
IF inv THEN
    Buffer := Value_Max - Buffer;
END_IF;

//Ограничение снизу
IF Buffer < Value_Min THEN
    Buffer := Value_Min;
END_IF;

//Ограничение сверху
IF Buffer > Value_Max THEN
    Buffer := Value_Max;
END_IF;

//Вывод значения
Result := Buffer;

END_FUNCTION

// System/FC/drv_Alarm
FUNCTION drv_Alarm : bool
VAR_INPUT
	Signal			:BOOL;		//alarm condition
	Reset			:BOOL;		//local reset command
END_VAR
VAR_IN_OUT
	Clock			:uni_Timer;
	Alarm			:BOOL;		//alarm signal
END_VAR

//Standart alarm control function
	//Conditions compelete
		IF Signal THEN
			Clock.plc.Start := TRUE;
		ELSE
			Clock.plc.Start := FALSE;
		END_IF
	//Alarm control
		IF Clock.plc.Q THEN
			Alarm := TRUE;
		END_IF
	//Alarm reset
		IF sys.All_Reset OR Reset THEN
			Clock.plc.Start := FALSE;
			Alarm := FALSE;
		END_IF

END_FUNCTION

// System/FC/drv_Time_S
FUNCTION drv_Time_S : bool
VAR_IN_OUT
	T			:Time_S;		//configuration and command struct for timer of seconds
END_VAR

// Timer with a multiplicity of 1 second
	IF T.CMD.plc.Start AND NOT T.CMD.plc.Reset THEN
		// Turn on
		IF T.AP < T.SP THEN
			IF NOT T.CMD.plc.Pause AND sys.pulse_1s THEN
				T.AP := T.AP + 1;
			END_IF;
			T.CMD.plc.Q := FALSE;
		ELSE
			// SP is achieved
			T.CMD.plc.Q := TRUE;
		END_IF;
	ELSE
		// Turn off and reset
		T.AP := 0;
		T.CMD.plc.Q := FALSE;
		T.CMD.plc.Reset := FALSE;
	END_IF;

END_FUNCTION

// Drivers/FB_sub/sub_Filter
FUNCTION_BLOCK sub_Filter
VAR_INPUT
	Start			:BOOL;		//Enable filter
	Signal			:REAL;		//Input value
	Filter_Type		:INT;		//Execution clock for filter: 0 = every cycle of PLC, 1 = 0.1s, 2 = 1s
	Filter_Lim 		:INT;		//Value of records in filter buffer
END_VAR
VAR_OUTPUT
	Result			:REAL;		//Median value for all measurments
END_VAR
VAR
	cnt				:INT;		//calculate actual measurments
	x				:INT;		//internal counter for shifting array elements
	exe				:BOOL;		//command to execution filtering cycle
	Summ			:REAL;		//Summary value of all array's values
	DATA			:ARRAY [0..100] OF REAL;
END_VAR

//limit
	IF Filter_Lim > 100 THEN
		Filter_Lim := 100;
	END_IF

//adding new entyty
IF Start AND (Filter_Type = 0 OR (Filter_Type = 1 AND sys.pulse_01s) OR (Filter_Type = 2 AND sys.pulse_1s)) THEN
    IF cnt < Filter_Lim THEN
        cnt := cnt + 1;
    END_IF;
	exe := TRUE;
ELSIF NOT Start THEN
	cnt := 0;
	Result := Signal;
END_IF;

//start cycle
IF exe THEN
	//read new value
	DATA[0] := Signal;
	Summ := 0.0;
	
	//limit values
	IF cnt > Filter_Lim THEN
		cnt := Filter_Lim;
	END_IF;
	
	//shifting array
	FOR x := Filter_Lim TO 1 BY -1 DO
		DATA[x] := DATA[x - 1];
		IF x <= cnt AND Start THEN
			Summ := Summ + DATA[x];
		END_IF;
	END_FOR;
	
	//calculate median values
	IF cnt > 0 THEN
		Result := Summ / cnt;
	ELSE
		Result := 0.0;
	END_IF;
	
	//end cycle
	exe := FALSE;
END_IF;

END_FUNCTION_BLOCK

// Drivers/FB_drv/drv_AO
FUNCTION_BLOCK drv_AO
VAR_INPUT
	Signal			:REAL;			//Control signal from algorythm
END_VAR	
VAR_IN_OUT
	CMD				:uni_CMD;		//Non-retain structure with command word
	cfg				:AO_cfg;		//Retain structure with settings
	state			:AO_state;		//Non-retain structure with states information
END_VAR
VAR_OUTPUT
	Result_R		:REAL;			//Analog output signal to PLC in REAL
	Result_I		:INT;			//Analog output signal to PLC in INT
END_VAR
VAR
	Value			:REAL;			//tmp value for calculating 
	support			:WORD;			//internal command buffer
	cnt				:INT;			//internal counter
	PT				:ARRAY [0..1] OF R_TRIG;
	NT				:ARRAY [0..1] OF F_TRIG;
	Filter			:sub_Filter;
END_VAR

//ANALOG OUTPUT
//control of typical analog command
// - Hz setpoint for motors
// - % setpoint for valves

//global commands
	//auto mode
		IF sys.All_Auto THEN
			CMD.plc.Manual := FALSE;
		END_IF;
	//global reset
		IF sys.All_Reset THEN
			CMD.plc.Reset := TRUE;
		END_IF
		
//convert data
	IF cfg.cfg.plc.use_NoEmrg THEN
		support.0 := FALSE;
	ELSE
		support.0 := sys.All_Block;
	END_IF
	
//device control
	drv_CMD(Emergency := support.0,
			CMD := CMD);
	//manual mode flag
		IF CMD.plc.Manual THEN sys.man.plc.xAO := TRUE; END_IF;
		IF NOT CMD.plc.Manual THEN
			cfg.SP_M := Signal;
		END_IF
	//disable
		IF NOT CMD.plc.Start_M THEN
			cfg.SP_M := 0;
		END_IF

//data convert to phisycal value scale
	drv_Converter(
		Signal := cfg.SP_M,
		Range := cfg.Range,
		Result => Value);
	
//convert data
	drv_Scale(
		Value := Value,
		Input_Type := cfg.Output_Type,
		Range := cfg.Range,
		Result => state.Signal);

//state signal transfer
	state.Result := Value;
	
//result
IF NOT cfg.cfg.plc.use_Sim THEN
	Result_R := Value;
	Result_I := REAL_TO_INT(Value);
ELSE
	Result_R := 0.0;
	Result_I := 0;
END_IF
	
//global state
	IF CMD.plc.Start_A THEN
		state.state.plc.xON := TRUE;
		state.state.plc.xOFF := FALSE;
	ELSE
		state.state.plc.xON := FALSE;
		state.state.plc.xOFF := TRUE;
	END_IF
	
//HMI light
	IF cfg.cfg.plc.use_Light THEN
		IF CMD.plc.Start_A THEN state.Status := 1; END_IF
		IF NOT CMD.plc.Start_A THEN state.Status := 0; END_IF
	ELSE
		state.Status := 0;
	END_IF
	
//reset
	IF CMD.plc.Reset THEN
		state.state.plc.Alarm := FALSE;
		CMD.plc.Alarm := FALSE;
		CMD.plc.Reset := FALSE;
	END_IF

END_FUNCTION_BLOCK

// Drivers/FB_drv/drv_DI
FUNCTION_BLOCK drv_DI
VAR_INPUT
	Signal			:BOOL;		//Physical input value, i.e. %IX0.6
END_VAR
VAR_IN_OUT
	CMD				:uni_CMD;	//Non-retain structure with command word
	cfg				:DI_cfg;	//Retain structure with settings
END_VAR
VAR_OUTPUT
	Result			:BOOL;		//Logical output value, used in algorythms
END_VAR
VAR
	Value			:BOOL;		//internal signal
	Clock			:ARRAY [0..1] OF Time_R;
END_VAR

//DIGITAL INPUT
//Signals from sensors, for example:
//	- keys
//	- sensors
//	- etc

//global commands
	//auto mode
		IF sys.All_Auto THEN
			CMD.plc.Manual := FALSE;
		END_IF;

//normal close mode
	IF cfg.cfg.plc.use_NC THEN
		Value := NOT Signal;
	ELSE
		Value := Signal;
	END_IF;
	
// chatter filter
	IF cfg.cfg.plc.use_Filter THEN
	//turn on
		IF cfg.SP_T_ON > 0 AND Value THEN
			Clock[1].CMD.plc.Start := TRUE;
			Clock[0].CMD.plc.Start := FALSE;
			IF Clock[1].CMD.plc.Q THEN
				CMD.plc.Start_A := Value;
			END_IF;
		ELSIF Value THEN
			CMD.plc.Start_A := TRUE;
			Clock[1].CMD.plc.Start := FALSE;
			Clock[0].CMD.plc.Start := FALSE;
		END_IF;
			
	//turn off
		IF cfg.SP_T_OFF > 0 AND NOT Value THEN
			Clock[1].CMD.plc.Start := FALSE;
			Clock[0].CMD.plc.Start := TRUE;
			IF Clock[0].CMD.plc.Q THEN
				CMD.plc.Start_A := Signal;
			END_IF;
		ELSIF NOT Value THEN
			CMD.plc.Start_A := FALSE;
			Clock[1].CMD.plc.Start := FALSE;
			Clock[0].CMD.plc.Start := FALSE;
		END_IF;
	ELSE
		CMD.plc.Start_A := Value;
	END_IF;

//device control
	drv_CMD(Emergency := FALSE,
		CMD := CMD);
	//manual mode flag
		IF CMD.plc.Manual THEN sys.man.plc.xDI := TRUE; END_IF;

//result for main logic
	Result := CMD.plc.Start_M;

//call timers
	Clock[0].SP := INT_TO_REAL(cfg.SP_T_OFF);
	Clock[1].SP := INT_TO_REAL(cfg.SP_T_ON);
	drv_Time_R (Clock[0]);
	drv_Time_R (Clock[1]);

END_FUNCTION_BLOCK

// System/FC/drv_Time_R
FUNCTION drv_Time_R : bool
VAR_IN_OUT
	T			:Time_R;			//configuration and command struct for timer of milliseconds
END_VAR

// Timer with a multiplicity of 1 second
		
	//time counting
	IF T.CMD.plc.Start AND NOT T.CMD.plc.Reset THEN
		// Turn on
			IF T.RTC = 0 THEN
				T.RTC := sys.UpTime_ms;
			END_IF
		//delta calculate
			IF NOT T.CMD.plc.Q THEN
				T.Delta := sys.UpTime_ms - T.RTC;
			END_IF;
		//delta control
		IF T.AP < T.SP THEN
			T.CMD.plc.Q := FALSE;
		ELSE
			T.CMD.plc.Q := TRUE;
		END_IF;
	ELSE
		// Turn off and reset
		T.AP := 0;
		T.RTC := 0;
		T.Delta := 0;
		T.CMD.plc.Q := FALSE;
		T.CMD.plc.Reset := FALSE;
	END_IF;
	
	//convert data
		T.AP := UDINT_TO_REAL(T.Delta) / 1000;
	
	//calculate time
		IF T.SP > 0 AND T.CMD.plc.Start THEN
			T.Percent := (T.AP / T.SP) * 100.0;
		ELSE
			T.Percent := 0;
		END_IF;

END_FUNCTION

// Drivers/FB_drv/drv_DO
FUNCTION_BLOCK drv_DO
VAR_INPUT
	Signal			:BOOL;			//Command in automation mode from algorythms
END_VAR
VAR_IN_OUT
	CMD				:uni_CMD;		//Non-retain structure with command word
	cfg				:DO_cfg;		//Retain structure with settings
END_VAR
VAR_OUTPUT
	Result			:BOOL;			//Phisical output signal, i.e. %QX2.4
END_VAR
VAR
	support			:WORD;			//internal command buffer
	PT				:ARRAY [0..1] OF R_TRIG;
	NT				:ARRAY [0..1] OF F_TRIG;
END_VAR

//DIGITAL OUTPUT
//control of primitive devices, for example
// - solenoid valve
// - signal for data exchange with another device
// - etc

//global commands
	//auto mode
		IF sys.All_Auto THEN
			CMD.plc.Manual := FALSE;
		END_IF;
	//simulation mode
		PT[0](CLK := sys.All_Sim);
		NT[0](CLK := sys.All_Sim);
		IF PT[0].Q THEN cfg.cfg.plc.use_Sim := TRUE; END_IF;
		IF NT[0].Q THEN cfg.cfg.plc.use_Sim := FALSE; END_IF;
		if cfg.cfg.plc.use_Sim then sys.sim.plc.xDI := TRUE; end_if;

//convert data
	CMD.plc.Start_A := Signal;
	IF cfg.cfg.plc.use_NoEmrg THEN
		support.0 := FALSE;
	ELSE
		support.0 := sys.All_Block;
	END_IF
	
//device control
	drv_CMD(Emergency := support.0,
		CMD := CMD);
	//manual mode flag
		IF CMD.plc.Manual THEN sys.man.plc.xDO := TRUE; END_IF;
		
//command transfer
	support.15 := CMD.plc.Start_M;

//normal close mode
	IF cfg.cfg.plc.use_NC AND NOT cfg.cfg.plc.use_Sim THEN
		Result := NOT support.15;
	ELSE
		Result := support.15;
	END_IF;
	
//simulation mode
	IF cfg.cfg.plc.use_Sim THEN
		Result := FALSE;
	END_IF;

END_FUNCTION_BLOCK

// Drivers/FB_drv/drv_DOA
FUNCTION_BLOCK drv_DOA
VAR_INPUT
	Signal			:BOOL;			//Command in automation mode from algorythms
END_VAR
VAR_IN_OUT
	CMD				:uni_CMD;		//Non-retain structure with command word
	cfg				:DO_cfg_ext;	//Retain structure with settings
END_VAR
VAR_OUTPUT
	Result			:BOOL;			//Phisical output signal, i.e. %QX2.4
END_VAR
VAR
	support			:WORD;			//internal command buffer
	cnt				:INT;			//internal counter
	PT				:ARRAY [0..1] OF R_TRIG;
	NT				:ARRAY [0..1] OF F_TRIG;
	Clock			:ARRAY [0..1] OF Time_R;
END_VAR

//DIGITAL OUTPUT
//control of primitive devices, for example
// - solenoid valve
// - signal for data exchange with another device
// - etc

//global commands
	//auto mode
		IF sys.All_Auto THEN
			CMD.plc.Manual := FALSE;
		END_IF;
	//simulation mode
		PT[0](CLK := sys.All_Sim);
		NT[0](CLK := sys.All_Sim);
		IF PT[0].Q THEN cfg.cfg.plc.use_Sim := TRUE; END_IF;
		IF NT[0].Q THEN cfg.cfg.plc.use_Sim := FALSE; END_IF;
		IF cfg.cfg.plc.use_Sim THEN sys.sim.plc.xDO := TRUE; END_IF;

//convert data
	CMD.plc.Start_A := Signal;
	IF cfg.cfg.plc.use_NoEmrg THEN
		support.0 := FALSE;
	ELSE
		support.0 := sys.All_Block;
	END_IF
	
//device control
	drv_CMD(Emergency := support.0,
		CMD := CMD);
	//manual mode flag
		IF CMD.plc.Manual THEN sys.man.plc.xDO := TRUE; END_IF;
		
//command transfer
	support.15 := CMD.plc.Start_M;
	IF NOT CMD.plc.Manual THEN
		cfg.SP_M := cfg.SP_A;
	END_IF
	
//timer control
	Clock[0].CMD.plc.Start := support.15;
	IF Clock[0].CMD.plc.Q THEN
		Clock[0].CMD.plc.Reset := TRUE;
	END_IF
	
//output control
	IF cfg.cfg.plc.use_PWM THEN
		IF support.15 THEN
			IF Clock[0].Percent < cfg.SP_M THEN
				support.14 := TRUE;
			ELSE
				support.14 := FALSE;
			END_IF
			IF Clock[0].Percent > cfg.SP_Max THEN
				support.14 := TRUE;
			END_IF
			IF Clock[0].Percent < cfg.SP_Min THEN
				support.14 := FALSE;
			END_IF
		ELSE
			support.14 := FALSE;
		END_IF
	ELSE
		support.14 := support.15;
	END_IF

//normal close mode
	IF cfg.cfg.plc.use_NC AND NOT cfg.cfg.plc.use_Sim THEN
		Result := NOT support.14;
	ELSE
		Result := support.14;
	END_IF;
	
//simulation mode
	IF cfg.cfg.plc.use_Sim THEN
		Result := FALSE;
	END_IF;
	
//call timers
	Clock[0].SP := cfg.SP_T;
	FOR cnt := 0 TO 1 DO
		drv_Time_R (Clock[cnt]);
	END_FOR

END_FUNCTION_BLOCK

// Drivers/FB_drv/drv_Flow
FUNCTION_BLOCK drv_Flow
VAR_INPUT
	Start			:BOOL;			//Start flow control
	Signal_DI		:BOOL;			//Discrete impulse from flowmeter
	Signal_AI		:REAL;			//Analog data from flowmeter
END_VAR	
VAR_IN_OUT
	CMD				:uni_CMD;		//Non-retain structure with command word
	cfg				:FE_cfg;		//Retain structure with settings
	state			:FE_state;		//Non-retain structure with states information
END_VAR
VAR_OUTPUT
	PreDone			:BOOL;			//PreSP reached
	Done			:BOOL;			//SP reached
	Result			:REAL;			//Signal from flowmeter
END_VAR
VAR
	AP				:REAL;			//Actual time for countimng
	AP_POU			:REAL;			//Last actual value for counting
	SW				:REAL;			//Start weight for control 
	Value			:REAL;			//tmp value for calculating 
	support			:WORD;			//internal command buffer
	cnt				:INT;			//internal counter
	PT				:ARRAY [0..1] OF R_TRIG;
	NT				:ARRAY [0..1] OF F_TRIG;
	Clock			:ARRAY [0..1] OF Time_X;
	Filter			:sub_Filter;
END_VAR

//FLOWMETER
//control of typical flowmeter control
// - value of source product
// - flowspeed
// - statistics
// - etc

//global commands
	//auto mode
		IF sys.All_Auto THEN
			CMD.plc.Manual := FALSE;
		END_IF;
	//global reset
		IF sys.All_Reset THEN
			CMD.plc.Reset := TRUE;
		END_IF
		
//device control
	CMD.plc.Start_A := Start;
	drv_CMD(Emergency := support.0,
			CMD := CMD);
	//manual mode flag
		IF CMD.plc.Manual THEN sys.man.plc.xFE := TRUE; END_IF;
	//reset counter
		PT[1](CLK := CMD.plc.Start_M);
		IF PT[1].Q THEN
			state.Last_AP := state.AP;
			state.AP := 0.0;
		END_IF

//impulse mode
	PT[0](CLK := Signal_DI);
	IF cfg.cfg.plc.use_DI AND NOT cfg.cfg.plc.use_FM THEN
		IF NOT cfg.cfg.plc.use_POU THEN
			//time reset
			IF PT[0].Q THEN
				Clock[0].CMD.plc.Reset := TRUE;
				AP := Clock[0].AP;
			END_IF 
			//time control
			Clock[0].CMD.plc.Start := CMD.plc.Start_M;
		ELSE
			IF NOT PT[0].Q THEN
				AP_POU := AP_POU + cfg.Clock;
				AP := AP_POU;
			ELSE
				AP_POU := 0;
			END_IF
		END_IF
	ELSE
		Clock[0].CMD.plc.Start := FALSE;
	END_IF
	
//signal's filter
	IF cfg.cfg.plc.use_DI THEN
		//discrete input filtering
		IF PT[0].Q THEN
			Filter(
				Start := CMD.plc.Start_M,
				Signal := AP,
				Filter_Type := 0,
				Filter_Lim := cfg.Filter_Lim,
				Result => Result);
		END_IF
	ELSE
		//analog input filtering
		Filter(
			Start := CMD.plc.Start_M AND cfg.cfg.plc.use_Filter,
			Signal := Signal_AI,
			Filter_Type := cfg.Filter_Type,
			Filter_Lim := cfg.Filter_Lim,
			Result => Result);
		IF NOT cfg.cfg.plc.use_Filter THEN
			Result := Value;
		END_IF
	END_IF

//weight mode
	IF  cfg.cfg.plc.use_FM THEN
		IF NOT support.2 AND CMD.plc.Start_M THEN
			SW := Signal_AI;
			support.2 := TRUE;
		END_IF
		IF support.2 THEN
			IF NOT cfg.cfg.plc.use_FM_Add THEN
				AP := SW - Signal_AI;
			ELSE
				AP := Signal_AI - SW;
			END_IF
		END_IF
	END_IF
	
//state signal transfer
	state.Result := Result;
	
//summary flow control
	IF CMD.plc.Start_M THEN
		//flow actual calculating
		IF cfg.cfg.plc.use_DI THEN
			//for DI
			state.AP := state.AP + cfg.Wieght;
		ELSIF NOT cfg.cfg.plc.use_FM THEN
			//for AI
			IF sys.pulse_01s THEN
				CASE cfg.Size_Time OF
					0:	state.AP := state.AP + Result / 3600 / 10;
					1:	state.AP := state.AP + Result / 60 / 10;
					2:	state.AP := state.AP + Result / 10;
				END_CASE 
			END_IF 
		END_IF 
		//pre-setpoint control
		IF state.AP >= cfg.PreSP THEN
			state.state.plc.Pos_Ok := TRUE;
		END_IF
		//setpoint control
		IF (state.AP >= (cfg.SP - cfg.DB)) THEN
			state.state.plc.Done := TRUE;
		END_IF
	END_IF
	
//deactivate control
	NT[0](CLK := CMD.plc.Start_M);
	IF NT[0].Q THEN
		state.state.plc.Pos_Ok := FALSE;
		state.state.plc.Done := FALSE;
	END_IF
	
//global state
	IF CMD.plc.Start_M THEN
		state.state.plc.xON := TRUE;
		state.state.plc.xOFF := FALSE;
	ELSE
		state.state.plc.xON := FALSE;
		state.state.plc.xOFF := TRUE;
	END_IF
	
//HMI light
	IF cfg.cfg.plc.use_Light THEN
		IF CMD.plc.Start_M AND NOT state.state.plc.Pos_Ok THEN state.Status := 3; END_IF
		IF CMD.plc.Start_M AND state.state.plc.Pos_Ok AND NOT state.state.plc.Done THEN state.Status := 2; END_IF
		IF state.state.plc.Done THEN state.Status := 1; END_IF
		IF NOT CMD.plc.Start_M THEN state.Status := 0; END_IF
	ELSE
		state.Status := 0;
	END_IF
	
//data transfer
	PreDone := state.state.plc.Pos_Ok;
	Done := state.state.plc.Done;
	
//reset
	IF CMD.plc.Reset THEN
		state.state.plc.Alarm := FALSE;
		CMD.plc.Alarm := FALSE;
		CMD.plc.Reset := FALSE;
	END_IF
	
//call timers
	FOR cnt := 0 TO 1 DO
		drv_Time_X (Clock[cnt]);
	END_FOR

END_FUNCTION_BLOCK

// System/FC/drv_Time_X
FUNCTION drv_Time_X : bool
VAR_IN_OUT
	T			:Time_X;			//configuration and command struct for timer of milliseconds
END_VAR

// Timer with a multiplicity of 1 second
		
	//time counting
	IF T.CMD.plc.Start AND NOT T.CMD.plc.Reset THEN
		// Turn on
			IF T.RTC = 0 THEN
				T.RTC := sys.UpTime_ms;
				T.Delta := 0;
			END_IF
		//delta calculate
			IF NOT T.CMD.plc.Q THEN
				T.Delta := sys.UpTime_ms - T.RTC;
			END_IF;
	ELSE
		// Turn off and reset
		T.RTC := 0;
		T.CMD.plc.Q := FALSE;
		T.CMD.plc.Reset := FALSE;
	END_IF;
	
	//convert data
		T.AP := UDINT_TO_REAL(T.Delta) / 1000;

END_FUNCTION

// Drivers/FB_drv/drv_M
FUNCTION_BLOCK drv_M
VAR_INPUT
	Signal			:BOOL;			//Command in automation mode from algorythms
	FB_QF			:BOOL;			//Physical input value, control feedback signal 'Ready' or NOT 'Alarm'
	FB_KM			:BOOL;			//Physical input value, control feedback signal 'In Work' OR 'Run'
END_VAR
VAR_IN_OUT
	CMD				:uni_CMD;		//Non-retain structure with command word
	cfg				:M_cfg;			//Retain structure with settings
	state			:M_state;		//Non-retain structure with states information
END_VAR
VAR_OUTPUT
	CMD_FW			:BOOL;			//Phisical output signal for start device, i.e. %QX2.4
	CMD_Low			:BOOL;			//Phisical output signal for speed control, i.e. %QX2.7 - optional
	Done			:BOOL;			//Device in work
END_VAR
VAR
	support			:WORD;			//internal command buffer
	cnt				:INT;			//internal counter
	alm				:ARRAY [0..3] OF BOOL;			//support word for transfer alarms
	PT				:ARRAY [0..1] OF R_TRIG;
	NT				:ARRAY [0..1] OF F_TRIG;
	Clock			:ARRAY [0..3] OF Time_S;
END_VAR

//MOTORS
//control of typical motors
// - ventitalitons
// - pumps
// - conveyors
// - etc

//global commands
	//start device
		IF cfg.cfg.plc.use_Signal THEN
			CMD.plc.Start_A := Signal;
		END_IF
	//auto mode
		IF sys.All_Auto THEN
			CMD.plc.Manual := FALSE;
			CMD.plc.Force := FALSE;
		END_IF;
	//simulation mode
		PT[0](CLK := sys.All_Sim);
		NT[0](CLK := sys.All_Sim);
		IF PT[0].Q THEN cfg.cfg.plc.use_Sim := TRUE; END_IF;
		IF NT[0].Q THEN cfg.cfg.plc.use_Sim := FALSE; END_IF;
		if cfg.cfg.plc.use_Sim then sys.sim.plc.xM := TRUE; end_if;
	//global reset
		IF sys.All_Reset THEN
			CMD.plc.Reset := TRUE;
		END_IF

//convert data
	IF cfg.cfg.plc.use_NoEmrg THEN
		support.0 := FALSE;
	ELSE
		support.0 := sys.All_Block;
		IF support.0 THEN
			state.Alarm.plc.alm_ES := TRUE;
			state.Status := 99;
		END_IF
	END_IF

//alarms without time control
	//QF control
		IF cfg.cfg.plc.use_QF THEN
			IF NOT FB_QF THEN
				state.Alarm.plc.alm_QF := TRUE;
				state.Status := 5;
			END_IF
		END_IF
	
//device control
	drv_CMD(Emergency := support.0,
		CMD := CMD);
	//manual mode flag
		IF CMD.plc.Manual THEN sys.man.plc.xM := TRUE; END_IF;
		
//delay turn on
	IF cfg.SP_T_Delay_ON > 0 AND NOT CMD.plc.Manual THEN
		IF CMD.plc.Start_M THEN
			Clock[0].CMD.plc.Start := TRUE;
			Clock[1].CMD.plc.Start := FALSE;
			IF Clock[0].CMD.plc.Q THEN
				support.1 := TRUE;
			END_IF
		ELSE
			Clock[0].CMD.plc.Start := FALSE;
		END_IF
	ELSE
		support.1 := CMD.plc.Start_M;
	END_IF

//delay turn off
	IF cfg.SP_T_Delay_OFF > 0 AND NOT CMD.plc.Manual THEN
		IF NOT CMD.plc.Start_M THEN
			Clock[1].CMD.plc.Start := TRUE;
			Clock[0].CMD.plc.Start := FALSE;
			IF Clock[1].CMD.plc.Q THEN
				support.1 := FALSE;
			END_IF
		ELSE
			Clock[1].CMD.plc.Start := FALSE;
		END_IF
	ELSE
		support.1 := CMD.plc.Start_M;
	END_IF
	
//Starting
	IF support.1 AND state.Status < 4 AND NOT cfg.cfg.plc.use_Sim THEN
		support.2 := TRUE;
		support.3 := FALSE;
		IF cfg.cfg.plc.use_KM THEN
			//starting in progress
			IF NOT Clock[2].CMD.plc.Q AND NOT FB_KM THEN
				state.Status := 2;
			END_IF
			//starting in fault
			IF Clock[2].CMD.plc.Q AND NOT FB_KM THEN
				state.Status := 6;
			END_IF
			//starting complieted
			IF FB_KM AND state.Status < 4THEN
				state.Status := 1;
			END_IF
		ELSE
			//succesfuly started
			state.Status := 1;
		END_IF
	END_IF
	
//Stopping
	IF NOT support.1 AND NOT cfg.cfg.plc.use_Sim THEN
		support.2 := FALSE;
		support.3 := TRUE;
		IF cfg.cfg.plc.use_KM THEN
			//stoping in progress
			IF NOT Clock[3].CMD.plc.Q AND FB_KM THEN
				state.Status := 3;
			END_IF
			//stoping in fault
			IF Clock[3].CMD.plc.Q AND FB_KM THEN
				state.Status := 7;
			END_IF
			//stoping complieted
			IF NOT FB_KM AND state.Status < 4 THEN
				state.Status := 0;
			END_IF
		ELSE
			//succesfuly stopped
			state.Status := 0;
		END_IF
	END_IF
		
//alarms with time control
	//start alarm control
		drv_Alarm(
			Signal := (support.2 AND NOT FB_KM),
			Reset := (CMD.plc.Reset OR cfg.cfg.plc.use_Sim),
			Clock := Clock[2].CMD,
			Alarm := alm[0]);
		state.Alarm.plc.alm_Start := alm[0];
	//stop alarm control
		drv_Alarm(
			Signal := (support.3 AND FB_KM),
			Reset := (CMD.plc.Reset OR cfg.cfg.plc.use_Sim),
			Clock := Clock[3].CMD,
			Alarm := alm[1]);
		state.Alarm.plc.alm_Stop := alm[1];	

//global alarm
	IF (state.Status > 4 OR state.Alarm.hmi > 0) AND NOT cfg.cfg.plc.use_Sim THEN
		state.state.plc.Alarm := TRUE;
		sys.alm.plc.xM := TRUE;
		CMD.plc.Alarm := TRUE;
	END_IF
			
//reset
	IF CMD.plc.Reset THEN
		IF state.Status > 4 THEN
			state.Status := 0;
		END_IF
		FOR cnt := 0 TO 6 DO
			Clock[cnt].CMD.plc.Reset := TRUE;
		END_FOR
		state.state.plc.Alarm := FALSE;
		state.Alarm.hmi := 0;
		CMD.plc.Alarm := FALSE;
		CMD.plc.Reset := FALSE;
	END_IF
	
//Simulation
	IF cfg.cfg.plc.use_Sim THEN
		IF support.1 THEN
			state.Status := 1;
		ELSE
			state.Status := 0;
		END_IF
	END_IF

//ON & OFF
	IF (FB_KM OR (CMD.plc.Start_M AND (cfg.cfg.plc.use_Sim OR NOT cfg.cfg.plc.use_KM))) AND state.Status < 4 THEN
		state.state.plc.xON := TRUE;	
		state.state.plc.xOFF := FALSE;	
	ELSIF (NOT FB_KM OR (NOT CMD.plc.Start_M AND (cfg.cfg.plc.use_Sim OR NOT cfg.cfg.plc.use_KM)))AND state.Status < 4 THEN
		state.state.plc.xON := FALSE;	
		state.state.plc.xOFF := TRUE;
	ELSE
		state.state.plc.xON := FALSE;	
		state.state.plc.xOFF := FALSE;
	END_IF
	
//Done
	Done := state.state.plc.xON;

//commands
	//turn on
		IF support.2 AND NOT state.state.plc.Pos_Ok THEN
			CMD_FW := TRUE;
			IF CMD.plc.LowSpeed THEN
				CMD_Low := TRUE;
			ELSE
				CMD_Low := FALSE;
			END_IF
		END_IF
	//turn off
		IF support.3 AND NOT state.state.plc.Pos_Ok THEN
			CMD_FW := FALSE;
			CMD_Low := FALSE;
		END_IF
	//shutdown
		IF cfg.cfg.plc.use_Sim THEN
			CMD_FW := FALSE;
			CMD_Low := FALSE;
			CMD.plc.Reset := TRUE;
		END_IF
	
//call timers
	Clock[0].SP := cfg.SP_T_Delay_ON;
	Clock[1].SP := cfg.SP_T_Delay_OFF;
	Clock[2].SP := cfg.SP_T_ON;
	Clock[3].SP := cfg.SP_T_OFF;
	FOR cnt := 0 TO 3 DO
		drv_Time_S (Clock[cnt]);
	END_FOR

END_FUNCTION_BLOCK

// Drivers/FB_drv/drv_MR
FUNCTION_BLOCK drv_MR
VAR_INPUT
	Signal			:BOOL;			//Command in automation mode from algorythms
	FB_QF			:BOOL;			//Physical input value, control feedback signal 'Ready' or NOT 'Alarm'
	FB_KM			:BOOL;			//Physical input value, control feedback signal 'In Work' OR 'Run'
END_VAR
VAR_IN_OUT
	CMD				:uni_CMD;		//Non-retain structure with command word
	cfg				:M_cfg;		//Retain structure with settings
	state			:M_state;	//Non-retain structure with states information
END_VAR
VAR_OUTPUT
	CMD_FW			:BOOL;			//Phisical output signal for start device forward, i.e. %QX2.4
	CMD_RV			:BOOL;			//Phisical output signal for start device reverse, i.e. %QX2.4
	CMD_Low			:BOOL;			//Phisical output signal for speed control, i.e. %QX2.7 - optional
	Done			:BOOL;			//Device in work
END_VAR
VAR
	support			:WORD;			//internal command buffer
	cnt				:INT;			//internal counter
	alm				:ARRAY [0..3] OF BOOL;			//support word for transfer alarms
	PT				:ARRAY [0..1] OF R_TRIG;
	NT				:ARRAY [0..1] OF F_TRIG;
	Clock			:ARRAY [0..3] OF Time_S;
END_VAR

//MOTORS
//control of typical motors
// - ventitalitons
// - pumps
// - conveyors
// - etc

//global commands
	//start device
		IF cfg.cfg.plc.use_Signal THEN
			CMD.plc.Start_A := Signal;
		END_IF
	//auto mode
		IF sys.All_Auto THEN
			CMD.plc.Manual := FALSE;
		END_IF;
	//simulation mode
		PT[0](CLK := sys.All_Sim);
		NT[0](CLK := sys.All_Sim);
		IF PT[0].Q THEN cfg.cfg.plc.use_Sim := TRUE; END_IF;
		IF NT[0].Q THEN cfg.cfg.plc.use_Sim := FALSE; END_IF;
		IF cfg.cfg.plc.use_Sim THEN sys.sim.plc.xM := TRUE; END_IF;
	//global reset
		IF sys.All_Reset THEN
			CMD.plc.Reset := TRUE;
		END_IF

//convert data
	IF cfg.cfg.plc.use_NoEmrg THEN
		support.0 := FALSE;
	ELSE
		support.0 := sys.All_Block;
		IF support.0 THEN
			state.Alarm.plc.alm_ES := TRUE;
			state.Status := 99;
		END_IF
	END_IF

//alarms without time control
	//QF control
		IF cfg.cfg.plc.use_QF THEN
			IF NOT FB_QF THEN
				state.Alarm.plc.alm_QF := TRUE;
				state.Status := 5;
			END_IF
		END_IF
	
//device control
	drv_CMD(Emergency := support.0,
		CMD := CMD);
	//manual mode flag
		IF CMD.plc.Manual THEN sys.man.plc.xM := TRUE; END_IF;
		
//delay turn on
	IF cfg.SP_T_Delay_ON > 0 AND NOT CMD.plc.Manual THEN
		IF CMD.plc.Start_M THEN
			Clock[0].CMD.plc.Start := TRUE;
			Clock[1].CMD.plc.Start := FALSE;
			IF Clock[0].CMD.plc.Q THEN
				support.1 := TRUE;
			END_IF
		ELSE
			Clock[0].CMD.plc.Start := FALSE;
		END_IF
	ELSE
		support.1 := CMD.plc.Start_M;
	END_IF

//delay turn off
	IF cfg.SP_T_Delay_OFF > 0 AND NOT CMD.plc.Manual THEN
		IF NOT CMD.plc.Start_M THEN
			Clock[1].CMD.plc.Start := TRUE;
			Clock[0].CMD.plc.Start := FALSE;
			IF Clock[1].CMD.plc.Q THEN
				support.1 := FALSE;
			END_IF
		ELSE
			Clock[1].CMD.plc.Start := FALSE;
		END_IF
	ELSE
		support.1 := CMD.plc.Start_M;
	END_IF
	
//Starting
	IF support.1 AND state.Status < 4 AND NOT cfg.cfg.plc.use_Sim THEN
		support.2 := TRUE;
		support.3 := FALSE;
		IF cfg.cfg.plc.use_KM THEN
			//starting in progress
			IF NOT Clock[2].CMD.plc.Q AND NOT FB_KM THEN
				state.Status := 2;
			END_IF
			//starting in fault
			IF Clock[2].CMD.plc.Q AND NOT FB_KM THEN
				state.Status := 6;
			END_IF
			//starting complieted
			IF FB_KM AND state.Status < 4THEN
				state.Status := 1;
			END_IF
		ELSE
			//succesfuly started
			state.Status := 1;
		END_IF
	END_IF
	
//Stopping
	IF NOT support.1 AND NOT cfg.cfg.plc.use_Sim THEN
		support.2 := FALSE;
		support.3 := TRUE;
		IF cfg.cfg.plc.use_KM THEN
			//stoping in progress
			IF NOT Clock[3].CMD.plc.Q AND FB_KM THEN
				state.Status := 3;
			END_IF
			//stoping in fault
			IF Clock[3].CMD.plc.Q AND FB_KM THEN
				state.Status := 7;
			END_IF
			//stoping complieted
			IF NOT FB_KM AND state.Status < 4 THEN
				state.Status := 0;
			END_IF
		ELSE
			//succesfuly stopped
			state.Status := 0;
		END_IF
	END_IF

//alarms with time control
	//start alarm control
		drv_Alarm(
			Signal := (support.2 AND NOT FB_KM),
			Reset := (CMD.plc.Reset OR cfg.cfg.plc.use_Sim),
			Clock := Clock[2].CMD,
			Alarm := alm[0]);
		state.Alarm.plc.alm_Start := alm[0];
	//stop alarm control
		drv_Alarm(
			Signal := (support.3 AND FB_KM),
			Reset := (CMD.plc.Reset OR cfg.cfg.plc.use_Sim),
			Clock := Clock[3].CMD,
			Alarm := alm[1]);
		state.Alarm.plc.alm_Stop := alm[1];	
		
//global alarm
	IF (state.Status > 4 OR state.Alarm.hmi > 0) AND NOT cfg.cfg.plc.use_Sim THEN
		state.state.plc.Alarm := TRUE;
		sys.alm.plc.xM := TRUE;
		CMD.plc.Alarm := TRUE;
	END_IF
			
//reset
	IF CMD.plc.Reset THEN
		IF state.Status > 4 THEN
			state.Status := 0;
		END_IF
		FOR cnt := 0 TO 6 DO
			Clock[cnt].CMD.plc.Reset := TRUE;
		END_FOR
		state.state.plc.Alarm := FALSE;
		state.Alarm.hmi := 0;
		CMD.plc.Alarm := FALSE;
		CMD.plc.Reset := FALSE;
	END_IF
	
//Simulation
	IF cfg.cfg.plc.use_Sim THEN
		IF support.1 THEN
			state.Status := 1;
		ELSE
			state.Status := 0;
		END_IF
	END_IF

//ON & OFF
	IF (FB_KM OR (CMD.plc.Start_M AND (cfg.cfg.plc.use_Sim OR NOT cfg.cfg.plc.use_KM))) AND state.Status < 4 THEN
		state.state.plc.xON := TRUE;	
		state.state.plc.xOFF := FALSE;	
	ELSIF (NOT FB_KM OR (NOT CMD.plc.Start_M AND (cfg.cfg.plc.use_Sim OR NOT cfg.cfg.plc.use_KM)))AND state.Status < 4 THEN
		state.state.plc.xON := FALSE;	
		state.state.plc.xOFF := TRUE;
	ELSE
		state.state.plc.xON := FALSE;	
		state.state.plc.xOFF := FALSE;
	END_IF
	
//Done
	Done := state.state.plc.xON;

//commands
	//turn on
		IF support.2 AND NOT state.state.plc.Pos_Ok THEN
			IF NOT CMD.plc.Direction THEN
				CMD_FW := TRUE;
				CMD_RV := FALSE;
			ELSE
				CMD_FW := FALSE;
				CMD_RV := TRUE;
			END_IF
			IF CMD.plc.LowSpeed THEN
				CMD_Low := TRUE;
			ELSE
				CMD_Low := FALSE;
			END_IF
		END_IF
	//turn off
		IF support.3 AND NOT state.state.plc.Pos_Ok THEN
			CMD_FW := FALSE;
			CMD_RV := FALSE;
			CMD_Low := FALSE;
		END_IF
	//shutdown
		IF cfg.cfg.plc.use_Sim THEN
			CMD_FW := FALSE;
			CMD_RV := FALSE;
			CMD_Low := FALSE;
			CMD.plc.Reset := TRUE;
		END_IF
	
//call timers
	Clock[0].SP := cfg.SP_T_Delay_ON;
	Clock[1].SP := cfg.SP_T_Delay_OFF;
	Clock[2].SP := cfg.SP_T_ON;
	Clock[3].SP := cfg.SP_T_OFF;
	FOR cnt := 0 TO 3 DO
		drv_Time_S (Clock[cnt]);
	END_FOR

END_FUNCTION_BLOCK

// Drivers/FB_drv/drv_V
FUNCTION_BLOCK drv_V
VAR_INPUT
	Signal			:BOOL;			//Command in automation mode from algorythms
	FB_QF			:BOOL;			//Physical input value, control feedback signal 'Ready' or NOT 'Alarm'
	FB_Open			:BOOL;			//Physical input value, control feedback signal 'Open'
	FB_Close		:BOOL;			//Physical input value, control feedback signal 'Close'
END_VAR
VAR_IN_OUT
	CMD				:uni_CMD;		//Non-retain structure with command word
	cfg				:V_cfg;			//Retain structure with settings
	state			:V_state;		//Non-retain structure with states information
END_VAR
VAR_OUTPUT
	CMD_Open		:BOOL;			//Phisical output signal for opening, i.e. %QX2.4
	CMD_Close		:BOOL;			//Phisical output signal for closing, i.e. %QX2.5
	CMD_Low			:BOOL;			//Phisical output signal for speed control, i.e. %QX2.7 - optional
	Done			:BOOL;			//Device is open
END_VAR
VAR
	support			:WORD;
	cnt				:INT;			//internal counter
	alm				:ARRAY [0..3] OF BOOL;			//support word for transfer alarms
	PT				:ARRAY [0..3] OF R_TRIG;
	NT				:ARRAY [0..1] OF F_TRIG;
	Clock			:ARRAY [0..3] OF Time_S;
END_VAR

//VALVES
//control of typical air and electrical valves
// - doors
// - dampers
// - valves
// - etc

//global commands
	//start device
		IF cfg.cfg.plc.use_Signal THEN
			CMD.plc.Start_A := Signal;
		END_IF
	//auto mode
		IF sys.All_Auto THEN
			CMD.plc.Manual := FALSE;
			CMD.plc.Force := FALSE;
		END_IF;
	//simulation mode
		PT[0](CLK := sys.All_Sim);
		NT[0](CLK := sys.All_Sim);
		IF PT[0].Q THEN cfg.cfg.plc.use_Sim := TRUE; END_IF;
		IF NT[0].Q THEN cfg.cfg.plc.use_Sim := FALSE; END_IF;
		IF cfg.cfg.plc.use_Sim THEN sys.sim.plc.xV := TRUE; END_IF;
	//global reset
		IF sys.All_Reset THEN
			CMD.plc.Reset := TRUE;
		END_IF

//convert data
	IF cfg.cfg.plc.use_NoEmrg THEN
		support.0 := FALSE;
	ELSE
		support.0 := sys.All_Block;
		IF support.0 THEN
			state.Alarm.plc.alm_ES := TRUE;
			state.Status := 99;
		END_IF
	END_IF

//alarms without time control
	//QF control
		IF cfg.cfg.plc.use_QF THEN
			IF NOT FB_QF THEN
				state.Alarm.plc.alm_QF := TRUE;
				state.Status := 5;
			END_IF
		END_IF
	
//device control
	drv_CMD(Emergency := support.0,
		CMD := CMD);
	//manual mode flag
		IF CMD.plc.Manual THEN sys.man.plc.xV := TRUE; END_IF;
		
//delay turn on
	IF cfg.SP_T_Delay_ON > 0 AND NOT CMD.plc.Manual THEN
		IF CMD.plc.Start_M THEN
			Clock[0].CMD.plc.Start := TRUE;
			Clock[1].CMD.plc.Start := FALSE;
			IF Clock[0].CMD.plc.Q THEN
				support.1 := TRUE;
			END_IF
		ELSE
			Clock[0].CMD.plc.Start := FALSE;
		END_IF
	ELSE
		support.1 := CMD.plc.Start_M;
	END_IF

//delay turn off
	IF cfg.SP_T_Delay_OFF > 0 AND NOT CMD.plc.Manual THEN
		IF NOT CMD.plc.Start_M THEN
			Clock[1].CMD.plc.Start := TRUE;
			Clock[0].CMD.plc.Start := FALSE;
			IF Clock[1].CMD.plc.Q THEN
				support.1 := FALSE;
			END_IF
		ELSE
			Clock[1].CMD.plc.Start := FALSE;
		END_IF
	ELSE
		support.1 := CMD.plc.Start_M;
	END_IF
	
//Opening
	IF support.1 AND state.Status < 4 AND NOT cfg.cfg.plc.use_Sim THEN
		IF cfg.cfg.plc.use_Air THEN
			support.2 := TRUE;
		ELSIF NOT cfg.cfg.plc.use_Air AND (NOT FB_Open OR NOT cfg.cfg.plc.use_FB_Open) THEN
			support.2 := TRUE;
		ELSE
			support.2 := FALSE;
		END_IF
		support.3 := FALSE;
		Clock[2].CMD.plc.Start := TRUE;
		Clock[3].CMD.plc.Start := FALSE;
		IF cfg.cfg.plc.use_FB_Open THEN
			//opening in progress
			IF NOT Clock[2].CMD.plc.Q AND NOT FB_Open THEN
				state.Status := 2;
			END_IF
			//opening in fault
			IF Clock[2].CMD.plc.Q AND NOT FB_Open AND NOT state.state.plc.Pos_Ok THEN
				state.Status := 6;
			END_IF
			//opening complieted
			IF FB_Open THEN
				state.Status := 1;
			END_IF
		ELSE
			//succesfuly
			state.Status := 1;
		END_IF
	END_IF
	
//Closing
	IF NOT support.1 AND NOT cfg.cfg.plc.use_Sim THEN
		support.2 := FALSE;
		IF cfg.cfg.plc.use_Air THEN
			support.3 := TRUE;
		ELSIF NOT cfg.cfg.plc.use_Air AND (NOT FB_Close OR NOT cfg.cfg.plc.use_FB_Close) THEN
			support.3 := TRUE;
		ELSE
			support.3 := FALSE;
		END_IF
		Clock[2].CMD.plc.Start := FALSE;
		Clock[3].CMD.plc.Start := TRUE;
		IF cfg.cfg.plc.use_FB_Close THEN
			//opening in progress
			IF NOT Clock[3].CMD.plc.Q AND NOT FB_Close THEN
				state.Status := 3;
			END_IF
			//opening in fault
			IF Clock[3].CMD.plc.Q AND NOT FB_Close AND NOT state.state.plc.Pos_Ok THEN
				state.Status := 7;
			END_IF
			//opening complieted
			IF FB_Close AND state.Status < 4 THEN
				state.Status := 0;
			END_IF
		ELSE
			//succesfuly
			state.Status := 0;
		END_IF
	END_IF
	
		
//alarms with time control
	//open alarm control
		drv_Alarm(
			Signal := (Clock[2].CMD.plc.Q AND NOT FB_Open AND NOT state.state.plc.Pos_Ok),
			Reset := (CMD.plc.Reset OR cfg.cfg.plc.use_Sim),
			Clock := Clock[2].CMD,
			Alarm := alm[0]);
		state.Alarm.plc.alm_Open := alm[0];
	//close alarm control
		drv_Alarm(
			Signal := (Clock[3].CMD.plc.Q AND NOT FB_Close AND NOT state.state.plc.Pos_Ok),
			Reset := (CMD.plc.Reset OR cfg.cfg.plc.use_Sim),
			Clock := Clock[3].CMD,
			Alarm := alm[1]);
		state.Alarm.plc.alm_Close := alm[1];	

//alarm control
	IF (state.Status > 4 OR state.Alarm.hmi > 0) AND NOT cfg.cfg.plc.use_Sim THEN
		state.state.plc.Alarm := TRUE;
		sys.alm.plc.xV := TRUE;
		CMD.plc.Alarm := TRUE;
	END_IF	
	
//disable close while alarm
	IF NOT cfg.cfg.plc.use_CWF AND state.state.plc.Alarm THEN
		support.2 := FALSE;
		support.3 := FALSE;
	END_IF
	
//reset
	IF CMD.plc.Reset THEN
		IF state.Status > 4 THEN
			state.Status := 0;
		END_IF
		FOR cnt := 0 TO 6 DO
			Clock[cnt].CMD.plc.Reset := TRUE;
		END_FOR
		state.state.plc.Alarm := FALSE;
		state.Alarm.hmi := 0;
		CMD.plc.Alarm := FALSE;
		CMD.plc.Reset := FALSE;
	END_IF

//Simulation
	IF cfg.cfg.plc.use_Sim THEN
		IF support.1 THEN
			state.Status := 1;
		ELSE
			state.Status := 0;
		END_IF
	END_IF
	
//ON & OFF, state
	IF (FB_Open OR (CMD.plc.Start_M AND (cfg.cfg.plc.use_Sim OR NOT cfg.cfg.plc.use_FB_Open))) AND state.Status < 4 THEN
		state.state.plc.xON := TRUE;	
		state.state.plc.xOFF := FALSE;	
	ELSIF (FB_Close OR (NOT CMD.plc.Start_M AND (cfg.cfg.plc.use_Sim OR NOT cfg.cfg.plc.use_FB_Close)))AND state.Status < 4 THEN
		state.state.plc.xON := FALSE;	
		state.state.plc.xOFF := TRUE;
	ELSE
		state.state.plc.xON := FALSE;	
		state.state.plc.xOFF := FALSE;
	END_IF
	
//Done
	Done := state.state.plc.xON;

//position control for once moving
	PT[1] (CLK := CMD.plc.Start_M);
	NT[1] (CLK := CMD.plc.Start_M);
	PT[2] (CLK := FB_Open); 
	PT[3] (CLK := FB_Close);
	IF cfg.cfg.plc.use_Once THEN
		IF PT[2].Q OR PT[3].Q THEN
			state.state.plc.Pos_Ok := TRUE;
		END_IF
		IF PT[1].Q OR NT[1].Q THEN
			state.state.plc.Pos_Ok := FALSE;
		END_IF
	ELSE
		state.state.plc.Pos_Ok := FALSE;
	END_IF
	
//commands
	//turn on
		IF support.2 AND NOT state.state.plc.Pos_Ok THEN
			CMD_Open := TRUE;
			CMD_Close := FALSE;
		END_IF
	//turn off
		IF support.3 AND NOT state.state.plc.Pos_Ok THEN
			IF NOT cfg.cfg.plc.use_Duo THEN
				CMD_Open := FALSE;
				CMD_Close := TRUE;
			ELSE
				CMD_Open := TRUE;
				CMD_Close := TRUE;
			END_IF
		END_IF
	//shutdown
		IF (NOT support.2 AND NOT support.3) OR state.state.plc.Pos_Ok OR cfg.cfg.plc.use_Sim THEN
			CMD_Open := FALSE;
			CMD_Close := FALSE;
		END_IF
	//low speed
		IF CMD_Open OR CMD_Close THEN
			IF CMD.plc.LowSpeed THEN
				CMD_Low := TRUE;
			ELSE
				CMD_Low := FALSE;
			END_IF
		END_IF
	
//call timers
	Clock[0].SP := cfg.SP_T_Delay_ON;
	Clock[1].SP := cfg.SP_T_Delay_OFF;
	Clock[2].SP := cfg.SP_T_ON;
	Clock[3].SP := cfg.SP_T_OFF;
	FOR cnt := 0 TO 3 DO
		drv_Time_S (Clock[cnt]);
	END_FOR

END_FUNCTION_BLOCK

// Drivers/FB_sub/sub_Axis_SP
FUNCTION sub_Axis_SP : bool
VAR_INPUT
	HMI				:list_Axis_SP;		//Значения, заданные пользователем
	Lim				:LREAL;
	C				:LREAL;
END_VAR
VAR_OUTPUT
	PLC				:list_Axis_SP;		//Значения, переданные программе
END_VAR

//Преобразование параметров движения с учётом коэффициента
	//Скорость
		PLC.Velocity := HMI.Velocity * C;
		IF PLC.Velocity > Lim THEN PLC.Velocity := Lim; END_IF
	//Ускорение
		PLC.Acceleration := HMI.Acceleration * C;
		IF PLC.Acceleration > Lim THEN PLC.Acceleration := Lim; END_IF
	//Замедление
		PLC.Deceleration := HMI.Deceleration * C;
		IF PLC.Deceleration > Lim THEN PLC.Deceleration := Lim; END_IF
	//Положение
		PLC.Position := HMI.Position * C;

END_FUNCTION

// Drivers/FB_sub/sub_Calibration
FUNCTION_BLOCK sub_Calibration
VAR_INPUT
	REQ				:BOOL;			//Request control
	Lim_FW			:BOOL;			//Limit switch forward
	Lim_RV			:BOOL;			//Limit switch rewers
	Mode			:BOOL;			//Claibration mode: 0 - RV->RW-RV, 1 - RW->RV-RW
END_VAR
VAR_OUTPUT
	CMD_FW			:BOOL;			//Command to move froward
	CMD_RV			:BOOL;			//Command to move reverse
	SP_FW			:REAL;			//Result time for forward moving
	SP_RV			:REAL;			//Result time for reverse moving
	state			:uni_state;		//Word of process state
END_VAR
VAR
	Step			:INT;			//step control for algorythm
	Value			:REAL;			//tmp value for calculating 
	support			:WORD;			//internal command buffer
	cnt				:INT;			//internal counter
	PT				:ARRAY [0..1] OF R_TRIG;
	NT				:ARRAY [0..1] OF F_TRIG;
	Clock			:ARRAY [0..2] OF Time_C;
END_VAR

//Algorithm for calibrating time for movement in two directions using limit switches

//global process control
IF NOT REQ THEN
	Step := 0;
END_IF
		
//Main process
CASE Step OF
	0:	//wait for start
		IF NOT REQ THEN
			CMD_FW := FALSE;
			CMD_RV := FALSE;
			state.plc.Busy := FALSE;
			state.plc.Done := FALSE;
			FOR cnt := 0 TO 2 DO
				Clock[cnt].One := 0.1;
				Clock[cnt].CMD.plc.Start := FALSE;
				Clock[cnt].CMD.plc.Pause := FALSE;
			END_FOR
		ELSE
			state.plc.Busy := TRUE;
			Step := 1;
		END_IF
	1:	//moving to start position
		IF NOT Mode THEN
			IF NOT Lim_FW THEN
				CMD_FW := TRUE;
			ELSE
				CMD_FW := FALSE;
				Step := 2;
			END_IF
		ELSE
			IF NOT Lim_RV THEN
				CMD_RV := TRUE;
			ELSE
				CMD_RV := FALSE;
				Step := 2;
			END_IF
		END_IF
	2:	//control time to 1st direction
		IF NOT Mode THEN
			CMD_FW := FALSE;
			CMD_RV := TRUE;
		ELSE
			CMD_FW := TRUE;
			CMD_RV := FALSE;
		END_IF
		Clock[1].CMD.plc.Start := TRUE;
		IF (Lim_FW AND Mode) OR (Lim_RV AND NOT Mode) THEN
			IF NOT Mode THEN
				SP_RV := Clock[1].AP;
			ELSE
				SP_FW := Clock[1].AP;
			END_IF
			Clock[1].CMD.plc.Pause := TRUE;
			CMD_FW := FALSE;
			CMD_RV := FALSE;
			Step := 3;
		END_IF
	3:	//control time to 2nd direction
		IF NOT Mode THEN
			CMD_FW := TRUE;
			CMD_RV := FALSE;
		ELSE
			CMD_FW := FALSE;
			CMD_RV := TRUE;
		END_IF
		Clock[2].CMD.plc.Start := TRUE;
		IF (Lim_FW AND NOT Mode) OR (Lim_RV AND Mode) THEN
			IF Mode THEN
				SP_RV := Clock[2].AP;
			ELSE
				SP_FW := Clock[2].AP;
			END_IF
			Clock[2].CMD.plc.Pause := TRUE;
			CMD_FW := FALSE;
			CMD_RV := FALSE;
			Step := 99;
		END_IF
	99:	//Final step
		state.plc.Busy := FALSE;
		state.plc.Done := TRUE;
END_CASE

//Control time move to 1st direction
drv_Time_C(
	Signal := sys.pulse_01s,
	T := Clock[1]);
	
//Control time move to 2nd direction
drv_Time_C(
	Signal := sys.pulse_01s,
	T := Clock[2]);

END_FUNCTION_BLOCK

// System/FC/drv_Time_C
FUNCTION drv_Time_C : bool
VAR_INPUT
	Signal 			:BOOL;			//signal from sensor or logical condition
END_VAR
VAR_IN_OUT
	T				:Time_C;		//configuration and command struct for counter
END_VAR

// Front signal control
	T.PT (CLK := Signal);
	
// Timer or counter with free multiplicity 
	IF T.CMD.plc.Start AND NOT T.CMD.plc.Reset THEN
		// Turn on
		IF NOT T.CMD.plc.Pause THEN
			IF T.PT.Q THEN
				T.AP := T.AP + T.One;
			END_IF;
		END_IF;
		//SP control
		IF T.AP < T.SP THEN
			// SP not achieved
			T.CMD.plc.Q := FALSE;
		ELSE
			// SP is achieved
			T.CMD.plc.Q := TRUE;
		END_IF;
	ELSE
		// Turn off and reset
		T.AP := 0.0;
		T.CMD.plc.Q := FALSE;
		T.CMD.plc.Reset := FALSE;
	END_IF;

// Progress control
	IF T.SP > 0 AND T.CMD.plc.Start THEN
		IF T.AP <= T.SP THEN
			T.Percent := (T.AP / T.SP) * 100.0;
		ELSE
			T.Percent := 100;
		END_IF
	ELSE
		T.Percent := 0.0;
	END_IF;

END_FUNCTION

// Drivers/FB_sub/sub_Slow
FUNCTION_BLOCK sub_Slow
VAR_IN_OUT
	REQ				:BOOL;			//Request control
	Signal			:REAL;
	cfg				:sub_Slow_cfg;
END_VAR
VAR_OUTPUT
	state			:uni_state;		//Word of process state
	Result			:REAL;
END_VAR
VAR
	Step			:INT;			//step control for algorythm
	Value			:REAL;			//tmp value for calculating 
	Delta			:REAL;			//delta between Signal and Result
	support			:WORD;			//internal command buffer
	cnt				:INT;			//internal counter
	PT				:ARRAY [0..1] OF R_TRIG;
	NT				:ARRAY [0..1] OF F_TRIG;
	Clock			:ARRAY [0..2] OF Time_R;
END_VAR

//Algorithm for slow control analogue value

//global process control
IF NOT cfg.cfg.plc.Enable THEN
	Result := Signal;
	Step := 0;
END_IF

//algorythm control
	PT[0](CLK := REQ);
	NT[0](CLK := REQ);

//Main process

IF Step = 0 THEN	//wait for start
	IF REQ THEN
		Step := 1;
	ELSIF NT[0].Q THEN
		Step := 20;
	ELSIF NOT REQ THEN
		Clock[1].CMD.plc.Start := FALSE;
		Clock[2].CMD.plc.Start := FALSE;
	END_IF
END_IF

IF Step = 1 THEN	//calculate delta
	Delta := Signal - Result;
	IF Delta > 0 THEN 
		state.plc.Done := FALSE;
		support.0 := FALSE;
		Step := 10;
 	ELSIF Delta < 0 THEN
		state.plc.Done := FALSE;
		support.0 := TRUE;
		Step := 20;
	ELSIF Delta = 0 THEN
		state.plc.Busy := FALSE;
		state.plc.Done := TRUE;
	END_IF;
	Delta := ABS(Delta);	
END_IF

IF Step = 10 THEN	//direction up
	//normal mode
	IF Delta > cfg.SP_Step_Up THEN
		Clock[1].CMD.plc.Start := TRUE;
		Clock[2].CMD.plc.Start := FALSE;
		IF Clock[1].CMD.plc.Q THEN
			Value := Value + cfg.SP_Step_Up;
			Clock[1].CMD.plc.Start := FALSE;
		END_IF
	ELSE
		Value := Signal;
	END_IF
	//forced up
	IF PT[0].Q AND cfg.cfg.plc.use_Force_Up THEN
		Value := Signal;
	END_IF
	//step control finished
	Step := 99;
END_IF

IF Step = 20 THEN	//direction down
	//normal mode
	IF Delta > cfg.SP_Step_Down THEN
		Clock[1].CMD.plc.Start := FALSE;
		Clock[2].CMD.plc.Start := TRUE;
		IF Clock[2].CMD.plc.Q THEN
			Value := Value - cfg.SP_Step_Down;
			Clock[2].CMD.plc.Start := FALSE;
		END_IF
	ELSE
		Value := Signal;
	END_IF
	//forced up
	IF NT[0].Q AND cfg.cfg.plc.use_Force_Down THEN
		Value := Signal;
	END_IF
	//step control finished
	Step := 99;
END_IF

IF Step = 99 THEN	//Finished step
	Step := 0;
END_IF

END_FUNCTION_BLOCK

// System/FC/drv_Time_01S
FUNCTION drv_Time_01S : bool
VAR_IN_OUT
	T			:Time_S;		//configuration and command struct for timer of seconds
END_VAR

// Timer with a multiplicity of 1 second
	IF T.CMD.plc.Start AND NOT T.CMD.plc.Reset THEN
		// Turn on
		IF T.AP < T.SP THEN
			IF NOT T.CMD.plc.Pause AND sys.pulse_01s THEN
				T.AP := T.AP + 1;
			END_IF;
			T.CMD.plc.Q := FALSE;
		ELSE
			// SP is achieved
			T.CMD.plc.Q := TRUE;
		END_IF;
	ELSE
		// Turn off and reset
		T.AP := 0;
		T.CMD.plc.Q := FALSE;
		T.CMD.plc.Reset := FALSE;
	END_IF;

END_FUNCTION
